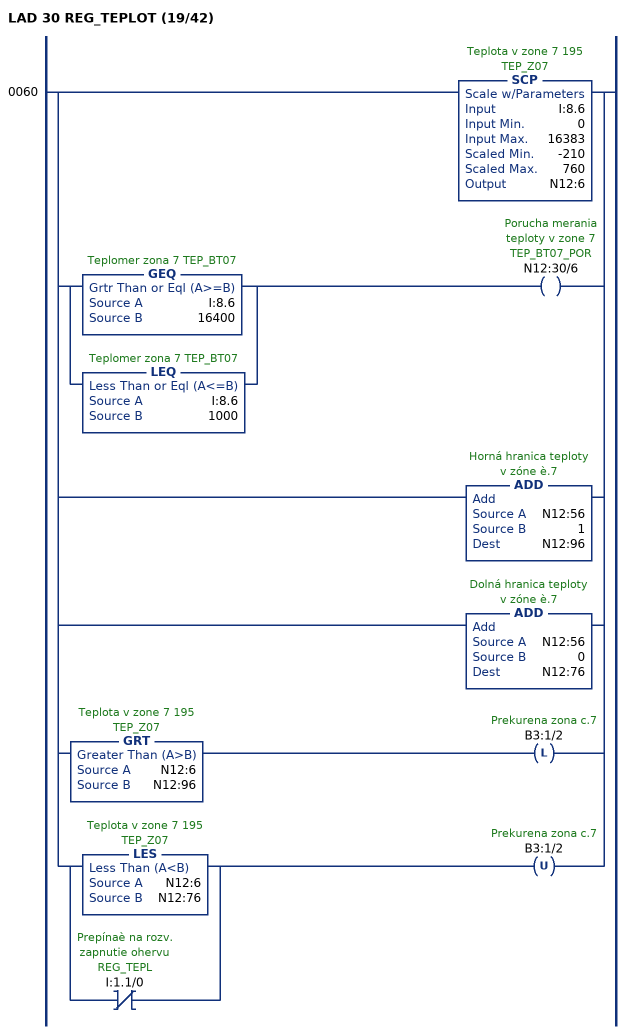
% Rung: 60 %
SOR BST SCP I:8.6 0 16383 -210 760 N12:6 NXB BST GEQ I:8.6 16400 NXB LEQ I:8.6 1000 BND OTE N12:30/6 NXB ADD N12:56 1 N12:96 NXB ADD N12:56 0 N12:76 NXB GRT N12:6 N12:96 OTL B3:1/2 NXB BST LES N12:6 N12:76 NXB XIO I:1.1/0 BND OTU B3:1/2 BND EOR
%   I:8.6  TEP_BT07  "Teplomer zona 7" %
%   N12:6  TEP_Z07  "Teplota v zone 7 195" %
%   N12:30/6  TEP_BT07_POR  "Porucha merania teploty v zone 7" %
%   N12:56  "Žiadaná teplota v zóne è.7" %
%   N12:96  "Horná hranica teploty v zóne è.7" %
%   N12:76  "Dolná hranica teploty v zóne è.7" %
%   B3:1/2  "Prekurena zona c.7" %
%   I:1.1/0  REG_TEPL  "Prepínaè na rozv. zapnutie ohervu" %

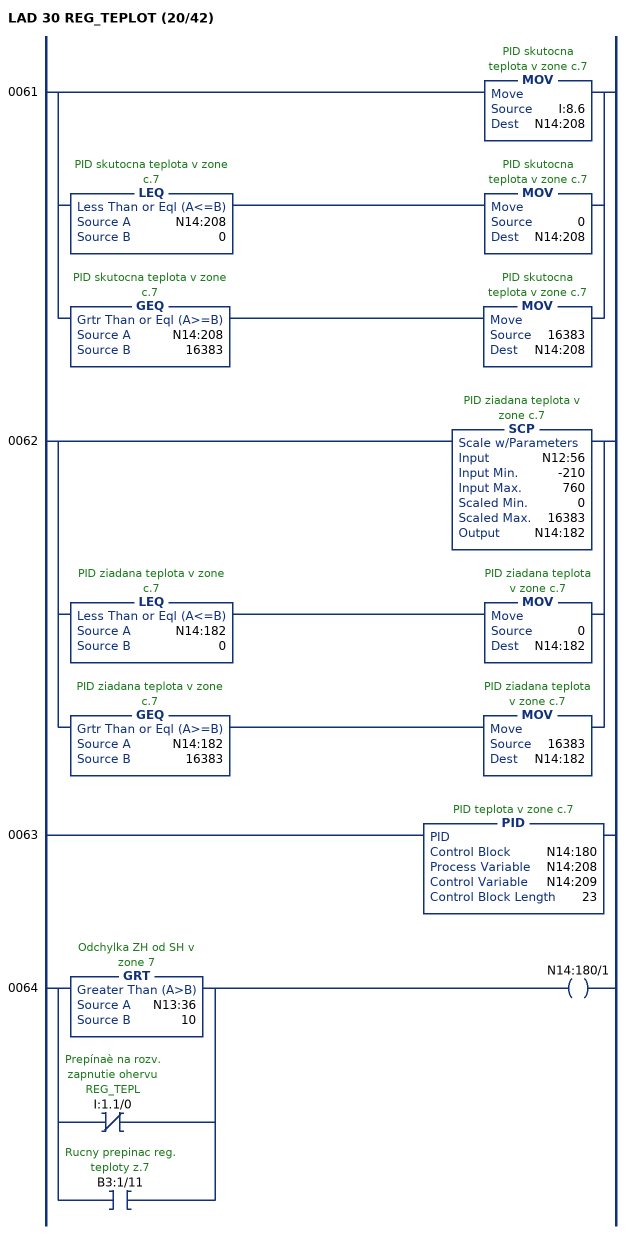
% Rung: 61 %
SOR BST MOV I:8.6 N14:208 NXB LEQ N14:208 0 MOV 0 N14:208 NXB GEQ N14:208 16383 MOV 16383 N14:208 BND EOR
%   I:8.6  TEP_BT07  "Teplomer zona 7" %
%   N14:208  "PID skutocna teplota v zone c.7" %
% Rung: 62 %
SOR BST SCP N12:56 -210 760 0 16383 N14:182 NXB LEQ N14:182 0 MOV 0 N14:182 NXB GEQ N14:182 16383 MOV 16383 N14:182 BND EOR
%   N12:56  "Žiadaná teplota v zóne è.7" %
%   N14:182  "PID ziadana teplota v zone c.7" %
% Rung: 63 %
SOR PID N14:180 N14:208 N14:209 23 EOR
%   N14:180  "PID teplota v zone c.7" %
%   N14:208  "PID skutocna teplota v zone c.7" %
% Rung: 64 %
SOR BST GRT N13:36 10 NXB XIO I:1.1/0 NXB XIC B3:1/11 BND OTE N14:180/1 EOR
%   N13:36  "Odchylka ZH od SH v zone 7" %
%   I:1.1/0  REG_TEPL  "Prepínaè na rozv. zapnutie ohervu" %
%   B3:1/11  "Rucny prepinac reg. teploty z.7" %

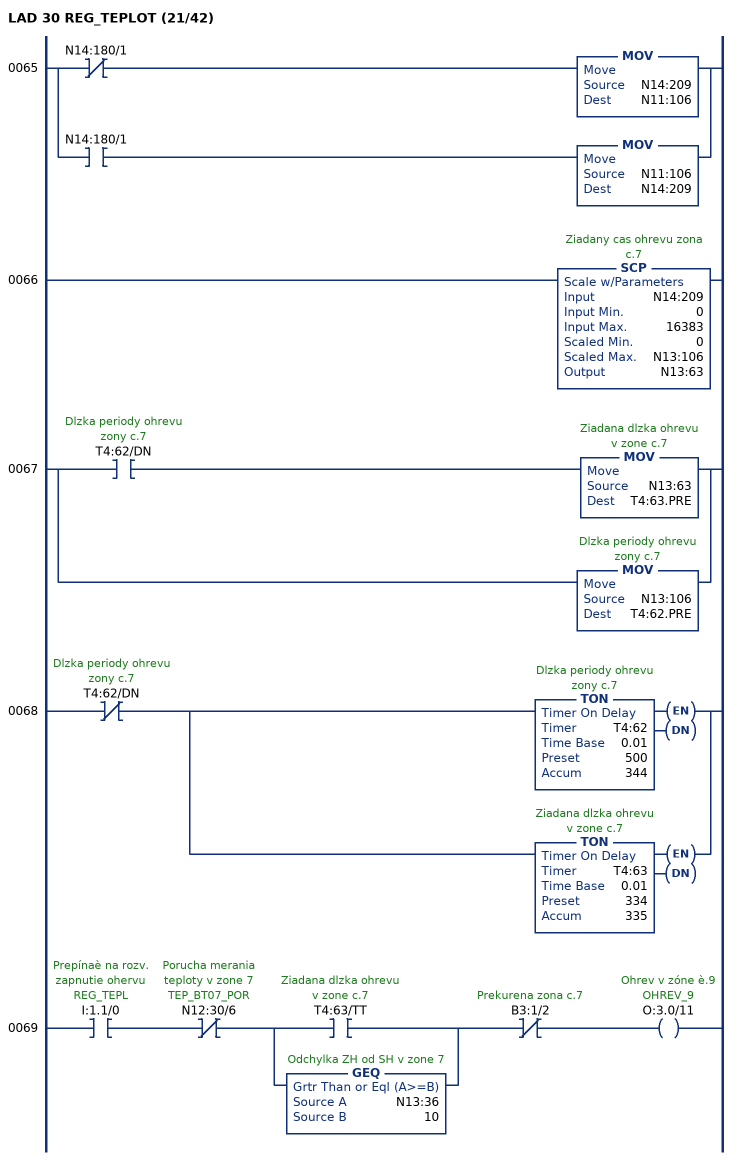
% Rung: 65 %
SOR BST XIO N14:180/1 MOV N14:209 N11:106 NXB XIC N14:180/1 MOV N11:106 N14:209 BND EOR
% Rung: 66 %
SOR SCP N14:209 0 16383 0 N13:106 N13:63 EOR
%   N13:63  "Ziadany cas ohrevu zona c.7" %
% Rung: 67 %
SOR BST XIC T4:62/DN MOV N13:63 T4:63.PRE NXB MOV N13:106 T4:62.PRE BND EOR
%   T4:62  "Dlzka periody ohrevu zony c.7" %
%   N13:63  "Ziadany cas ohrevu zona c.7" %
%   T4:63  "Ziadana dlzka ohrevu v zone c.7" %
% Rung: 68 %
SOR XIO T4:62/DN BST TON T4:62 0.01 500 344 NXB TON T4:63 0.01 334 335 BND EOR
%   T4:62  "Dlzka periody ohrevu zony c.7" %
%   T4:63  "Ziadana dlzka ohrevu v zone c.7" %
% Rung: 69 %
SOR XIC I:1.1/0 XIO N12:30/6 BST XIC T4:63/TT NXB GEQ N13:36 10 BND XIO B3:1/2 OTE O:3.0/11 EOR
%   I:1.1/0  REG_TEPL  "Prepínaè na rozv. zapnutie ohervu" %
%   N12:30/6  TEP_BT07_POR  "Porucha merania teploty v zone 7" %
%   T4:63  "Ziadana dlzka ohrevu v zone c.7" %
%   N13:36  "Odchylka ZH od SH v zone 7" %
%   B3:1/2  "Prekurena zona c.7" %
%   O:3.0/11  OHREV_9  "Ohrev v zóne è.9" %

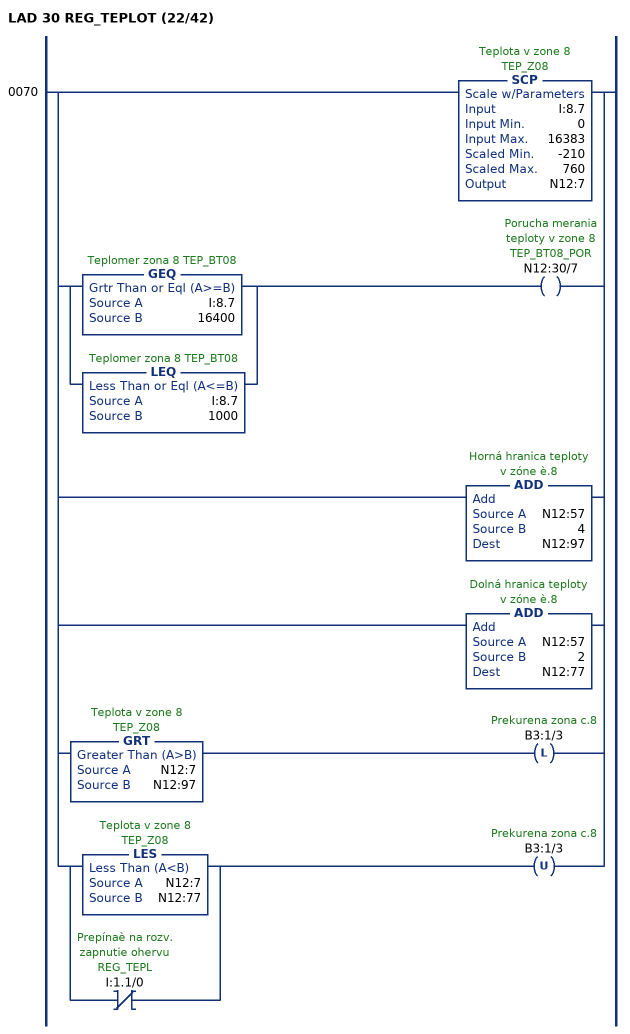
% Rung: 70 %
SOR BST SCP I:8.7 0 16383 -210 760 N12:7 NXB BST GEQ I:8.7 16400 NXB LEQ I:8.7 1000 BND OTE N12:30/7 NXB ADD N12:57 4 N12:97 NXB ADD N12:57 2 N12:77 NXB GRT N12:7 N12:97 OTL B3:1/3 NXB BST LES N12:7 N12:77 NXB XIO I:1.1/0 BND OTU B3:1/3 BND EOR
%   I:8.7  TEP_BT08  "Teplomer zona 8" %
%   N12:7  TEP_Z08  "Teplota v zone 8" %
%   N12:30/7  TEP_BT08_POR  "Porucha merania teploty v zone 8" %
%   N12:57  "Žiadaná teplota v zóne è.8" %
%   N12:97  "Horná hranica teploty v zóne è.8" %
%   N12:77  "Dolná hranica teploty v zóne è.8" %
%   B3:1/3  "Prekurena zona c.8" %
%   I:1.1/0  REG_TEPL  "Prepínaè na rozv. zapnutie ohervu" %

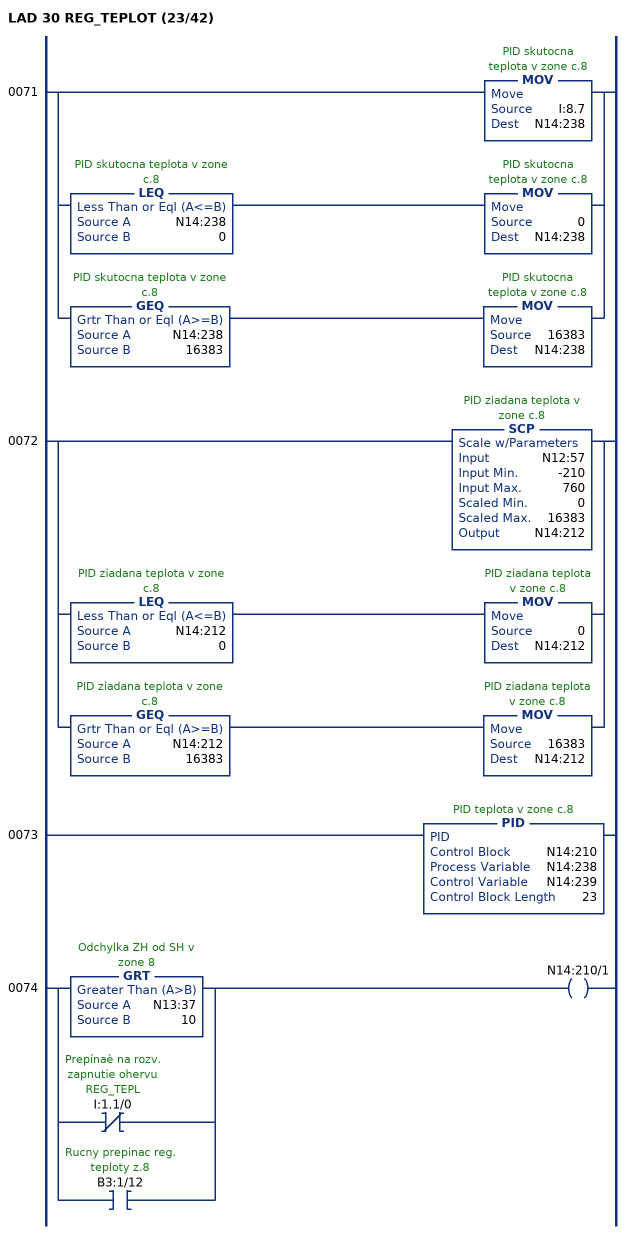
% Rung: 71 %
SOR BST MOV I:8.7 N14:238 NXB LEQ N14:238 0 MOV 0 N14:238 NXB GEQ N14:238 16383 MOV 16383 N14:238 BND EOR
%   I:8.7  TEP_BT08  "Teplomer zona 8" %
%   N14:238  "PID skutocna teplota v zone c.8" %
% Rung: 72 %
SOR BST SCP N12:57 -210 760 0 16383 N14:212 NXB LEQ N14:212 0 MOV 0 N14:212 NXB GEQ N14:212 16383 MOV 16383 N14:212 BND EOR
%   N12:57  "Žiadaná teplota v zóne è.8" %
%   N14:212  "PID ziadana teplota v zone c.8" %
% Rung: 73 %
SOR PID N14:210 N14:238 N14:239 23 EOR
%   N14:210  "PID teplota v zone c.8" %
%   N14:238  "PID skutocna teplota v zone c.8" %
% Rung: 74 %
SOR BST GRT N13:37 10 NXB XIO I:1.1/0 NXB XIC B3:1/12 BND OTE N14:210/1 EOR
%   N13:37  "Odchylka ZH od SH v zone 8" %
%   I:1.1/0  REG_TEPL  "Prepínaè na rozv. zapnutie ohervu" %
%   B3:1/12  "Rucny prepinac reg. teploty z.8" %

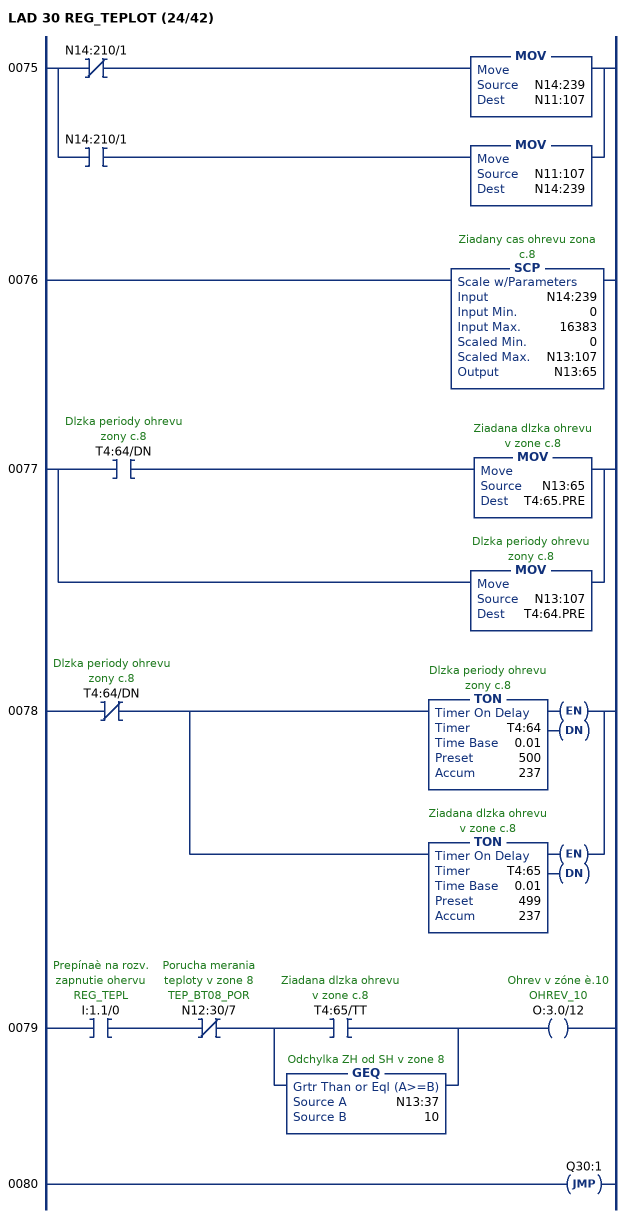
% Rung: 75 %
SOR BST XIO N14:210/1 MOV N14:239 N11:107 NXB XIC N14:210/1 MOV N11:107 N14:239 BND EOR
% Rung: 76 %
SOR SCP N14:239 0 16383 0 N13:107 N13:65 EOR
%   N13:65  "Ziadany cas ohrevu zona c.8" %
% Rung: 77 %
SOR BST XIC T4:64/DN MOV N13:65 T4:65.PRE NXB MOV N13:107 T4:64.PRE BND EOR
%   T4:64  "Dlzka periody ohrevu zony c.8" %
%   N13:65  "Ziadany cas ohrevu zona c.8" %
%   T4:65  "Ziadana dlzka ohrevu v zone c.8" %
% Rung: 78 %
SOR XIO T4:64/DN BST TON T4:64 0.01 500 237 NXB TON T4:65 0.01 499 237 BND EOR
%   T4:64  "Dlzka periody ohrevu zony c.8" %
%   T4:65  "Ziadana dlzka ohrevu v zone c.8" %
% Rung: 79 %
SOR XIC I:1.1/0 XIO N12:30/7 BST XIC T4:65/TT NXB GEQ N13:37 10 BND OTE O:3.0/12 EOR
%   I:1.1/0  REG_TEPL  "Prepínaè na rozv. zapnutie ohervu" %
%   N12:30/7  TEP_BT08_POR  "Porucha merania teploty v zone 8" %
%   T4:65  "Ziadana dlzka ohrevu v zone c.8" %
%   N13:37  "Odchylka ZH od SH v zone 8" %
%   O:3.0/12  OHREV_10  "Ohrev v zóne è.10" %
% Rung: 80 %
SOR JMP Q30:1 EOR

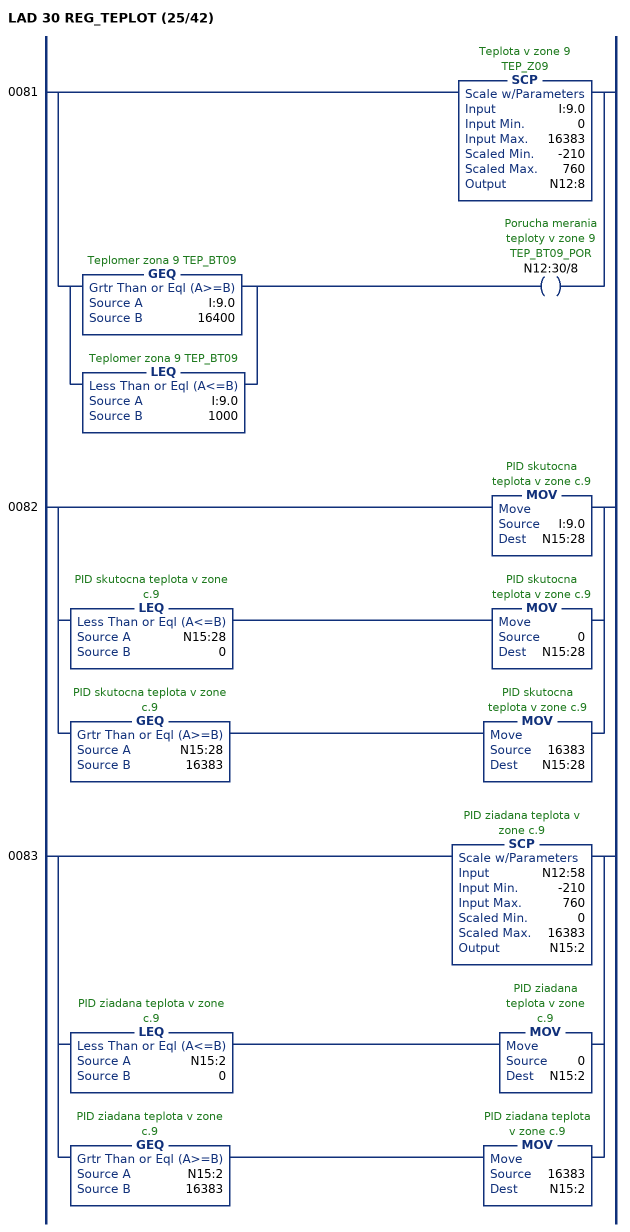
% Rung: 81 %
SOR BST SCP I:9.0 0 16383 -210 760 N12:8 NXB BST GEQ I:9.0 16400 NXB LEQ I:9.0 1000 BND OTE N12:30/8 BND EOR
%   I:9.0  TEP_BT09  "Teplomer zona 9" %
%   N12:8  TEP_Z09  "Teplota v zone 9" %
%   N12:30/8  TEP_BT09_POR  "Porucha merania teploty v zone 9" %
% Rung: 82 %
SOR BST MOV I:9.0 N15:28 NXB LEQ N15:28 0 MOV 0 N15:28 NXB GEQ N15:28 16383 MOV 16383 N15:28 BND EOR
%   I:9.0  TEP_BT09  "Teplomer zona 9" %
%   N15:28  "PID skutocna teplota v zone c.9" %
% Rung: 83 %
SOR BST SCP N12:58 -210 760 0 16383 N15:2 NXB LEQ N15:2 0 MOV 0 N15:2 NXB GEQ N15:2 16383 MOV 16383 N15:2 BND EOR
%   N12:58  "Žiadaná teplota v zóne è.9" %
%   N15:2  "PID ziadana teplota v zone c.9" %

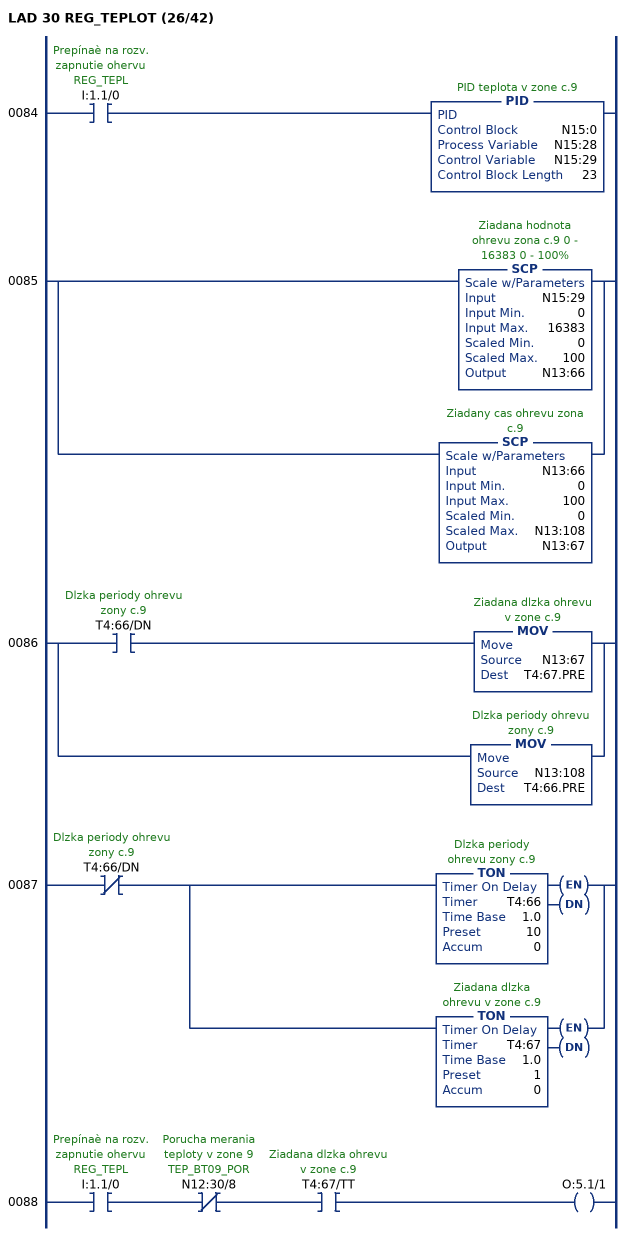
% Rung: 84 %
SOR XIC I:1.1/0 PID N15:0 N15:28 N15:29 23 EOR
%   I:1.1/0  REG_TEPL  "Prepínaè na rozv. zapnutie ohervu" %
%   N15:0  "PID teplota v zone c.9" %
%   N15:28  "PID skutocna teplota v zone c.9" %
% Rung: 85 %
SOR BST SCP N15:29 0 16383 0 100 N13:66 NXB SCP N13:66 0 100 0 N13:108 N13:67 BND EOR
%   N13:66  "Ziadana hodnota ohrevu zona c.9 0 - 16383 0 - 100%" %
%   N13:67  "Ziadany cas ohrevu zona c.9" %
% Rung: 86 %
SOR BST XIC T4:66/DN MOV N13:67 T4:67.PRE NXB MOV N13:108 T4:66.PRE BND EOR
%   T4:66  "Dlzka periody ohrevu zony c.9" %
%   N13:67  "Ziadany cas ohrevu zona c.9" %
%   T4:67  "Ziadana dlzka ohrevu v zone c.9" %
% Rung: 87 %
SOR XIO T4:66/DN BST TON T4:66 1.0 10 0 NXB TON T4:67 1.0 1 0 BND EOR
%   T4:66  "Dlzka periody ohrevu zony c.9" %
%   T4:67  "Ziadana dlzka ohrevu v zone c.9" %
% Rung: 88 %
SOR XIC I:1.1/0 XIO N12:30/8 XIC T4:67/TT OTE O:5.1/1 EOR
%   I:1.1/0  REG_TEPL  "Prepínaè na rozv. zapnutie ohervu" %
%   N12:30/8  TEP_BT09_POR  "Porucha merania teploty v zone 9" %
%   T4:67  "Ziadana dlzka ohrevu v zone c.9" %

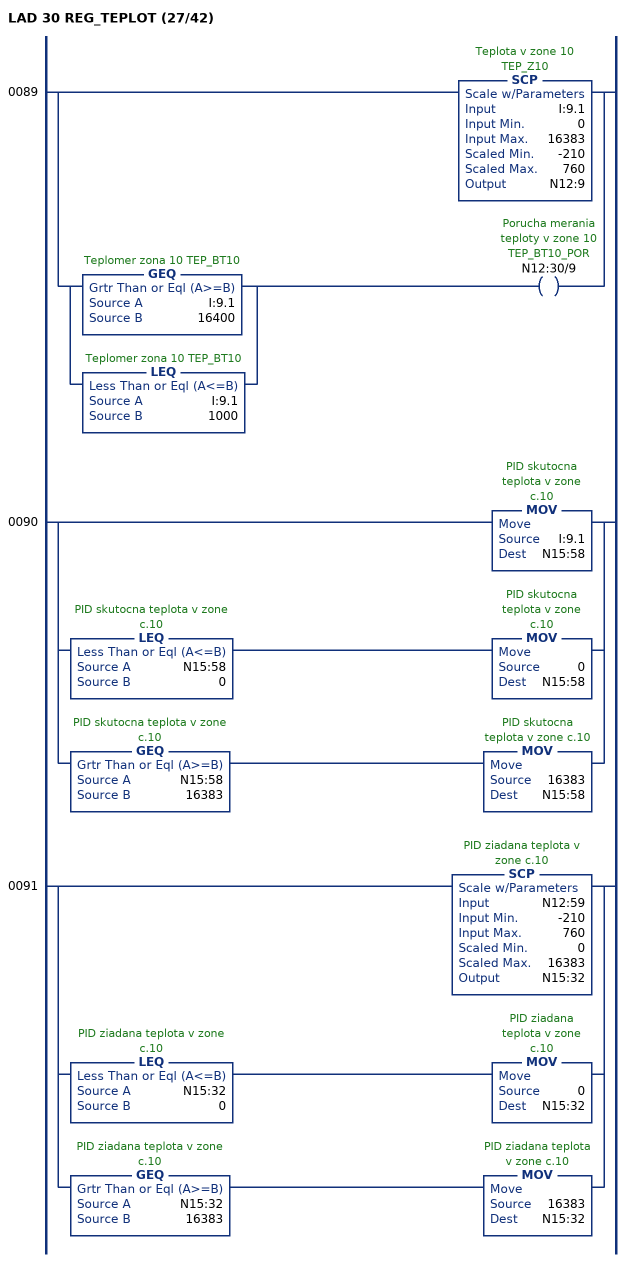
% Rung: 89 %
SOR BST SCP I:9.1 0 16383 -210 760 N12:9 NXB BST GEQ I:9.1 16400 NXB LEQ I:9.1 1000 BND OTE N12:30/9 BND EOR
%   I:9.1  TEP_BT10  "Teplomer zona 10" %
%   N12:9  TEP_Z10  "Teplota v zone 10" %
%   N12:30/9  TEP_BT10_POR  "Porucha merania teploty v zone 10" %
% Rung: 90 %
SOR BST MOV I:9.1 N15:58 NXB LEQ N15:58 0 MOV 0 N15:58 NXB GEQ N15:58 16383 MOV 16383 N15:58 BND EOR
%   I:9.1  TEP_BT10  "Teplomer zona 10" %
%   N15:58  "PID skutocna teplota v zone c.10" %
% Rung: 91 %
SOR BST SCP N12:59 -210 760 0 16383 N15:32 NXB LEQ N15:32 0 MOV 0 N15:32 NXB GEQ N15:32 16383 MOV 16383 N15:32 BND EOR
%   N12:59  "Žiadaná teplota v zóne è.10" %
%   N15:32  "PID ziadana teplota v zone c.10" %

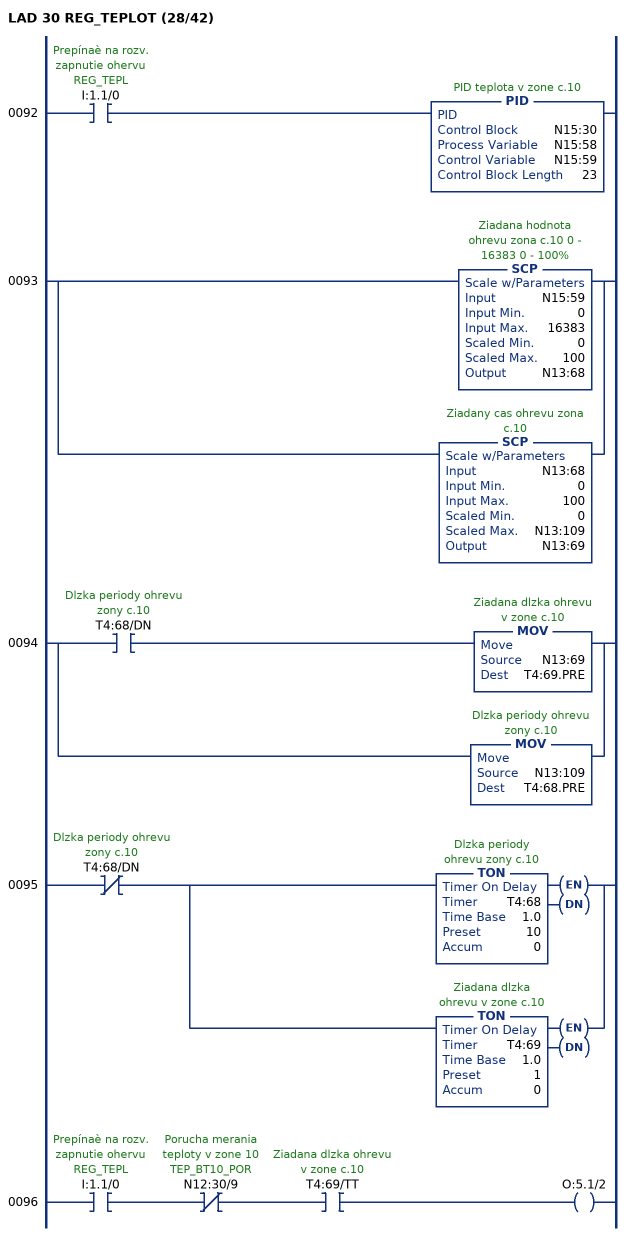
% Rung: 92 %
SOR XIC I:1.1/0 PID N15:30 N15:58 N15:59 23 EOR
%   I:1.1/0  REG_TEPL  "Prepínaè na rozv. zapnutie ohervu" %
%   N15:30  "PID teplota v zone c.10" %
%   N15:58  "PID skutocna teplota v zone c.10" %
% Rung: 93 %
SOR BST SCP N15:59 0 16383 0 100 N13:68 NXB SCP N13:68 0 100 0 N13:109 N13:69 BND EOR
%   N13:68  "Ziadana hodnota ohrevu zona c.10 0 - 16383 0 - 100%" %
%   N13:69  "Ziadany cas ohrevu zona c.10" %
% Rung: 94 %
SOR BST XIC T4:68/DN MOV N13:69 T4:69.PRE NXB MOV N13:109 T4:68.PRE BND EOR
%   T4:68  "Dlzka periody ohrevu zony c.10" %
%   N13:69  "Ziadany cas ohrevu zona c.10" %
%   T4:69  "Ziadana dlzka ohrevu v zone c.10" %
% Rung: 95 %
SOR XIO T4:68/DN BST TON T4:68 1.0 10 0 NXB TON T4:69 1.0 1 0 BND EOR
%   T4:68  "Dlzka periody ohrevu zony c.10" %
%   T4:69  "Ziadana dlzka ohrevu v zone c.10" %
% Rung: 96 %
SOR XIC I:1.1/0 XIO N12:30/9 XIC T4:69/TT OTE O:5.1/2 EOR
%   I:1.1/0  REG_TEPL  "Prepínaè na rozv. zapnutie ohervu" %
%   N12:30/9  TEP_BT10_POR  "Porucha merania teploty v zone 10" %
%   T4:69  "Ziadana dlzka ohrevu v zone c.10" %

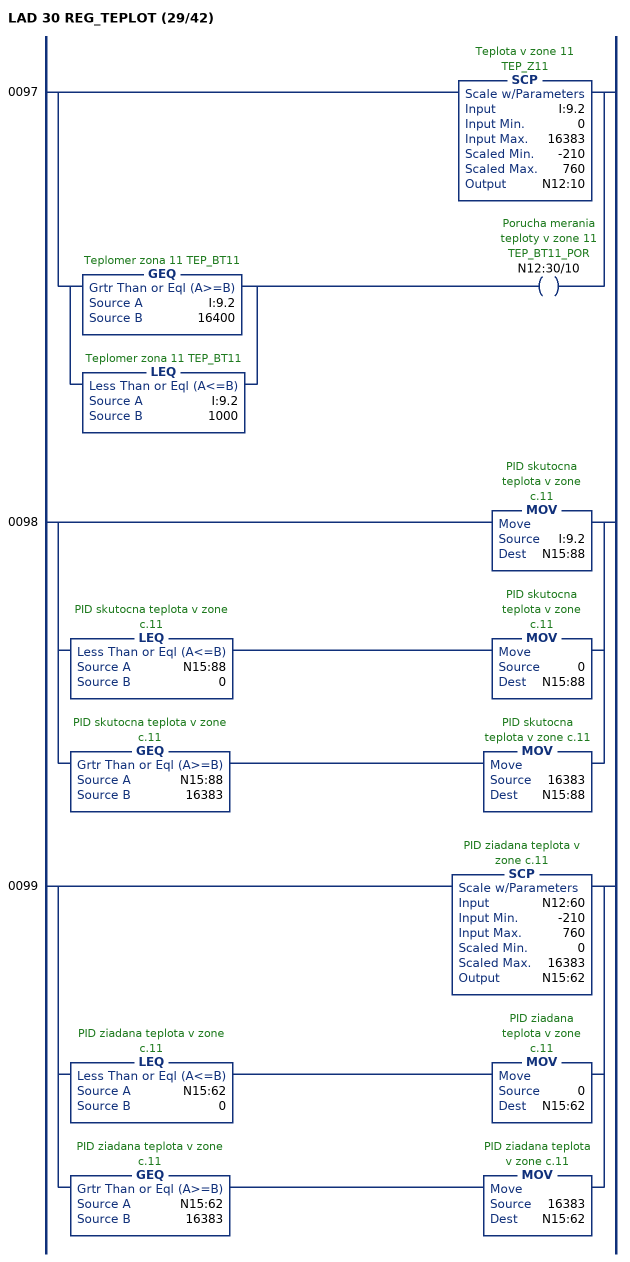
% Rung: 97 %
SOR BST SCP I:9.2 0 16383 -210 760 N12:10 NXB BST GEQ I:9.2 16400 NXB LEQ I:9.2 1000 BND OTE N12:30/10 BND EOR
%   I:9.2  TEP_BT11  "Teplomer zona 11" %
%   N12:10  TEP_Z11  "Teplota v zone 11" %
%   N12:30/10  TEP_BT11_POR  "Porucha merania teploty v zone 11" %
% Rung: 98 %
SOR BST MOV I:9.2 N15:88 NXB LEQ N15:88 0 MOV 0 N15:88 NXB GEQ N15:88 16383 MOV 16383 N15:88 BND EOR
%   I:9.2  TEP_BT11  "Teplomer zona 11" %
%   N15:88  "PID skutocna teplota v zone c.11" %
% Rung: 99 %
SOR BST SCP N12:60 -210 760 0 16383 N15:62 NXB LEQ N15:62 0 MOV 0 N15:62 NXB GEQ N15:62 16383 MOV 16383 N15:62 BND EOR
%   N12:60  "Žiadaná teplota v zóne è.11" %
%   N15:62  "PID ziadana teplota v zone c.11" %

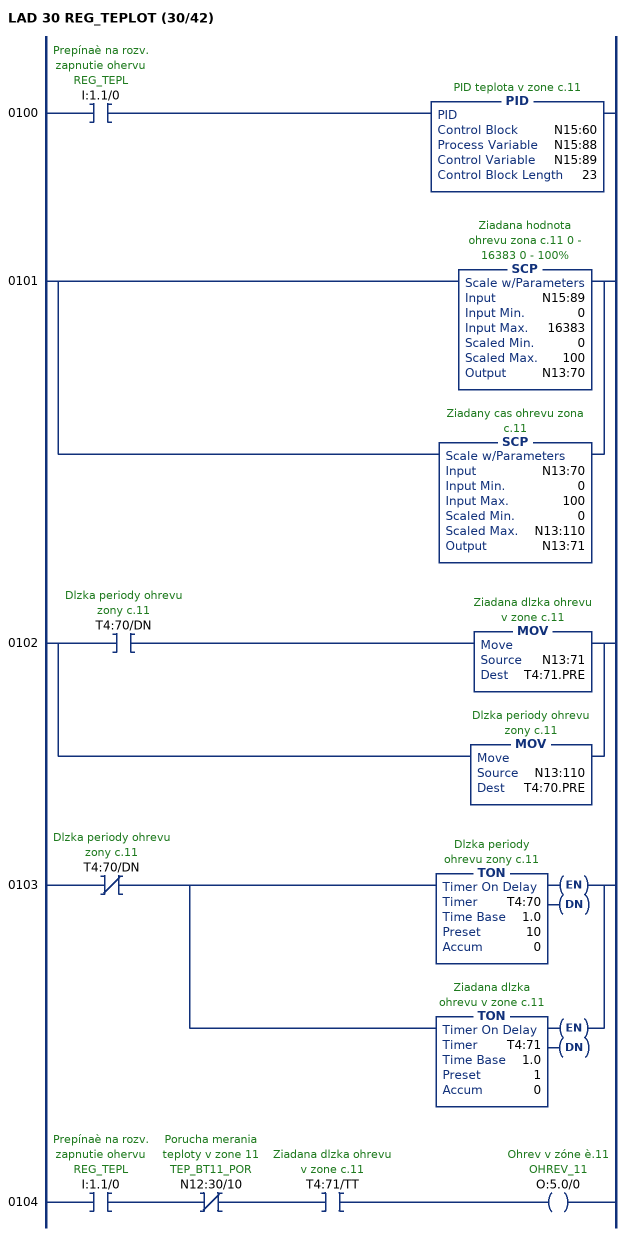
% Rung: 100 %
SOR XIC I:1.1/0 PID N15:60 N15:88 N15:89 23 EOR
%   I:1.1/0  REG_TEPL  "Prepínaè na rozv. zapnutie ohervu" %
%   N15:60  "PID teplota v zone c.11" %
%   N15:88  "PID skutocna teplota v zone c.11" %
% Rung: 101 %
SOR BST SCP N15:89 0 16383 0 100 N13:70 NXB SCP N13:70 0 100 0 N13:110 N13:71 BND EOR
%   N13:70  "Ziadana hodnota ohrevu zona c.11 0 - 16383 0 - 100%" %
%   N13:71  "Ziadany cas ohrevu zona c.11" %
% Rung: 102 %
SOR BST XIC T4:70/DN MOV N13:71 T4:71.PRE NXB MOV N13:110 T4:70.PRE BND EOR
%   T4:70  "Dlzka periody ohrevu zony c.11" %
%   N13:71  "Ziadany cas ohrevu zona c.11" %
%   T4:71  "Ziadana dlzka ohrevu v zone c.11" %
% Rung: 103 %
SOR XIO T4:70/DN BST TON T4:70 1.0 10 0 NXB TON T4:71 1.0 1 0 BND EOR
%   T4:70  "Dlzka periody ohrevu zony c.11" %
%   T4:71  "Ziadana dlzka ohrevu v zone c.11" %
% Rung: 104 %
SOR XIC I:1.1/0 XIO N12:30/10 XIC T4:71/TT OTE O:5.0/0 EOR
%   I:1.1/0  REG_TEPL  "Prepínaè na rozv. zapnutie ohervu" %
%   N12:30/10  TEP_BT11_POR  "Porucha merania teploty v zone 11" %
%   T4:71  "Ziadana dlzka ohrevu v zone c.11" %
%   O:5.0/0  OHREV_11  "Ohrev v zóne è.11" %

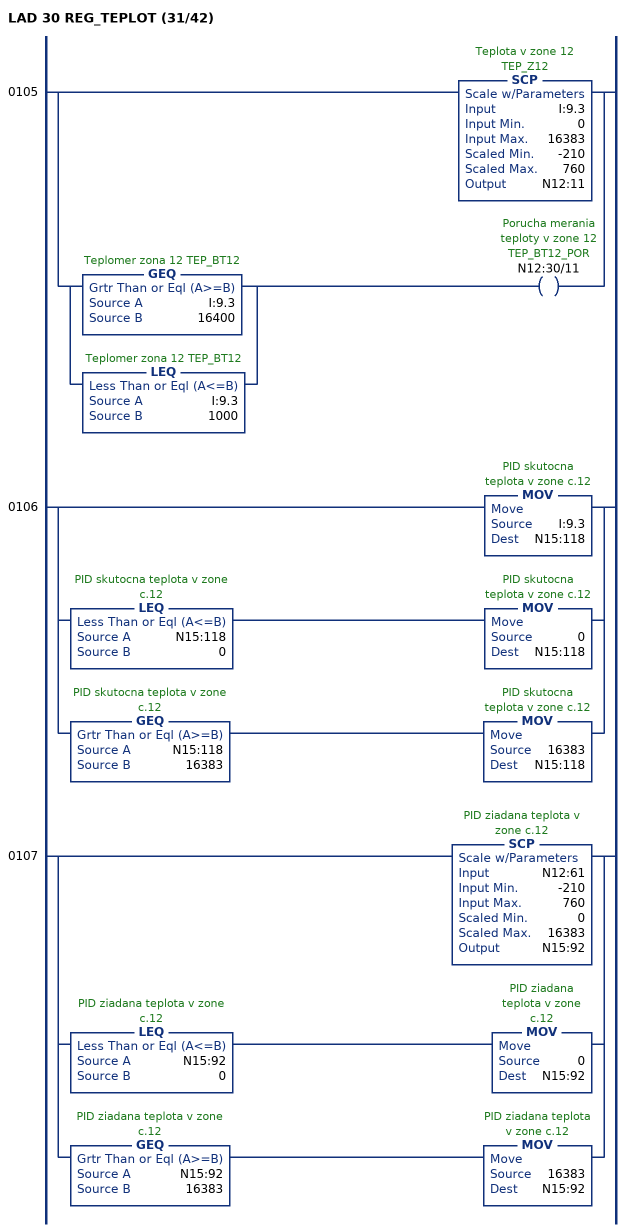
% Rung: 105 %
SOR BST SCP I:9.3 0 16383 -210 760 N12:11 NXB BST GEQ I:9.3 16400 NXB LEQ I:9.3 1000 BND OTE N12:30/11 BND EOR
%   I:9.3  TEP_BT12  "Teplomer zona 12" %
%   N12:11  TEP_Z12  "Teplota v zone 12" %
%   N12:30/11  TEP_BT12_POR  "Porucha merania teploty v zone 12" %
% Rung: 106 %
SOR BST MOV I:9.3 N15:118 NXB LEQ N15:118 0 MOV 0 N15:118 NXB GEQ N15:118 16383 MOV 16383 N15:118 BND EOR
%   I:9.3  TEP_BT12  "Teplomer zona 12" %
%   N15:118  "PID skutocna teplota v zone c.12" %
% Rung: 107 %
SOR BST SCP N12:61 -210 760 0 16383 N15:92 NXB LEQ N15:92 0 MOV 0 N15:92 NXB GEQ N15:92 16383 MOV 16383 N15:92 BND EOR
%   N12:61  "Žiadaná teplota v zóne è.12" %
%   N15:92  "PID ziadana teplota v zone c.12" %

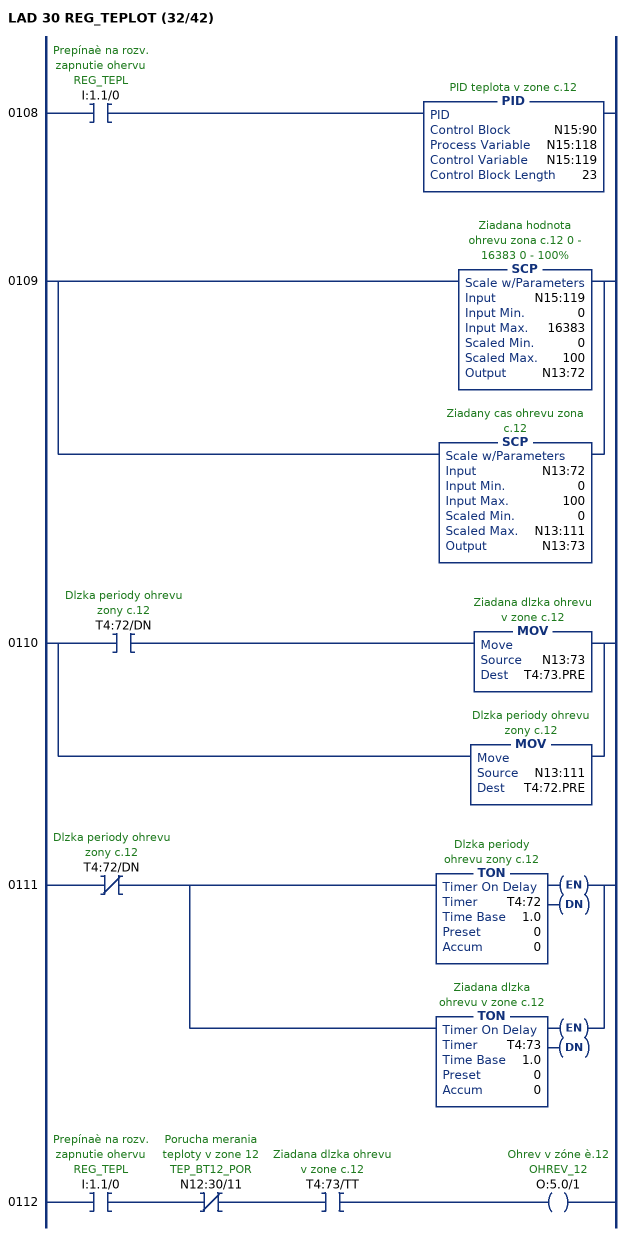
% Rung: 108 %
SOR XIC I:1.1/0 PID N15:90 N15:118 N15:119 23 EOR
%   I:1.1/0  REG_TEPL  "Prepínaè na rozv. zapnutie ohervu" %
%   N15:90  "PID teplota v zone c.12" %
%   N15:118  "PID skutocna teplota v zone c.12" %
% Rung: 109 %
SOR BST SCP N15:119 0 16383 0 100 N13:72 NXB SCP N13:72 0 100 0 N13:111 N13:73 BND EOR
%   N13:72  "Ziadana hodnota ohrevu zona c.12 0 - 16383 0 - 100%" %
%   N13:73  "Ziadany cas ohrevu zona c.12" %
% Rung: 110 %
SOR BST XIC T4:72/DN MOV N13:73 T4:73.PRE NXB MOV N13:111 T4:72.PRE BND EOR
%   T4:72  "Dlzka periody ohrevu zony c.12" %
%   N13:73  "Ziadany cas ohrevu zona c.12" %
%   T4:73  "Ziadana dlzka ohrevu v zone c.12" %
% Rung: 111 %
SOR XIO T4:72/DN BST TON T4:72 1.0 0 0 NXB TON T4:73 1.0 0 0 BND EOR
%   T4:72  "Dlzka periody ohrevu zony c.12" %
%   T4:73  "Ziadana dlzka ohrevu v zone c.12" %
% Rung: 112 %
SOR XIC I:1.1/0 XIO N12:30/11 XIC T4:73/TT OTE O:5.0/1 EOR
%   I:1.1/0  REG_TEPL  "Prepínaè na rozv. zapnutie ohervu" %
%   N12:30/11  TEP_BT12_POR  "Porucha merania teploty v zone 12" %
%   T4:73  "Ziadana dlzka ohrevu v zone c.12" %
%   O:5.0/1  OHREV_12  "Ohrev v zóne è.12" %

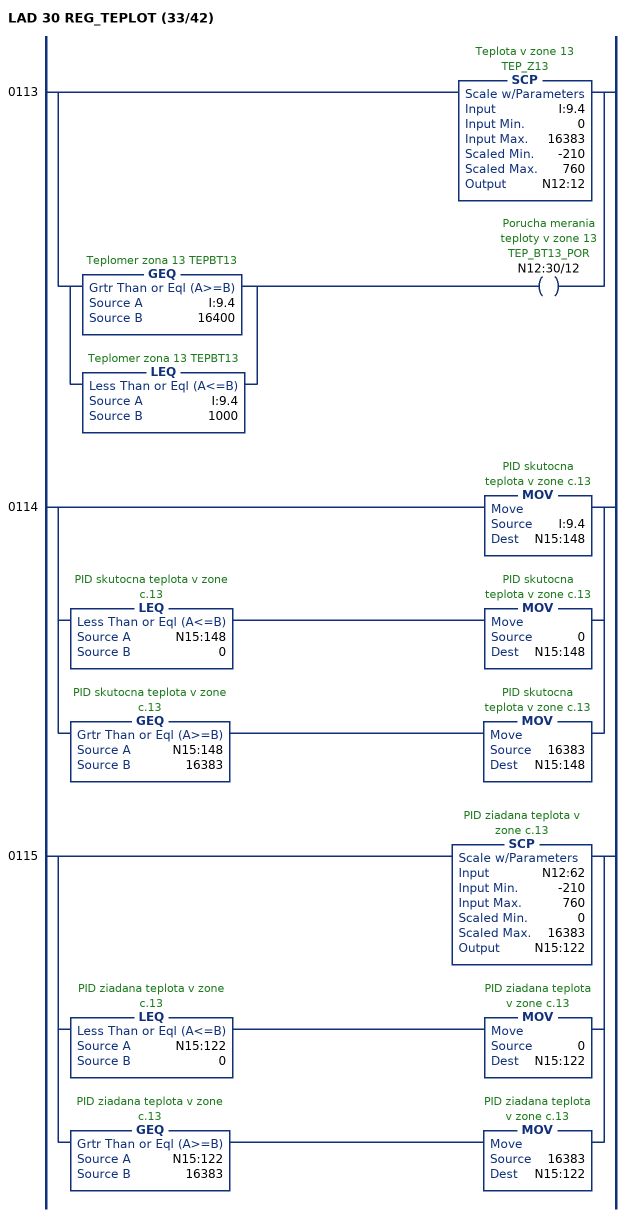
% Rung: 113 %
SOR BST SCP I:9.4 0 16383 -210 760 N12:12 NXB BST GEQ I:9.4 16400 NXB LEQ I:9.4 1000 BND OTE N12:30/12 BND EOR
%   I:9.4  TEPBT13  "Teplomer zona 13" %
%   N12:12  TEP_Z13  "Teplota v zone 13" %
%   N12:30/12  TEP_BT13_POR  "Porucha merania teploty v zone 13" %
% Rung: 114 %
SOR BST MOV I:9.4 N15:148 NXB LEQ N15:148 0 MOV 0 N15:148 NXB GEQ N15:148 16383 MOV 16383 N15:148 BND EOR
%   I:9.4  TEPBT13  "Teplomer zona 13" %
%   N15:148  "PID skutocna teplota v zone c.13" %
% Rung: 115 %
SOR BST SCP N12:62 -210 760 0 16383 N15:122 NXB LEQ N15:122 0 MOV 0 N15:122 NXB GEQ N15:122 16383 MOV 16383 N15:122 BND EOR
%   N12:62  "Žiadaná teplota v zóne è.13" %
%   N15:122  "PID ziadana teplota v zone c.13" %

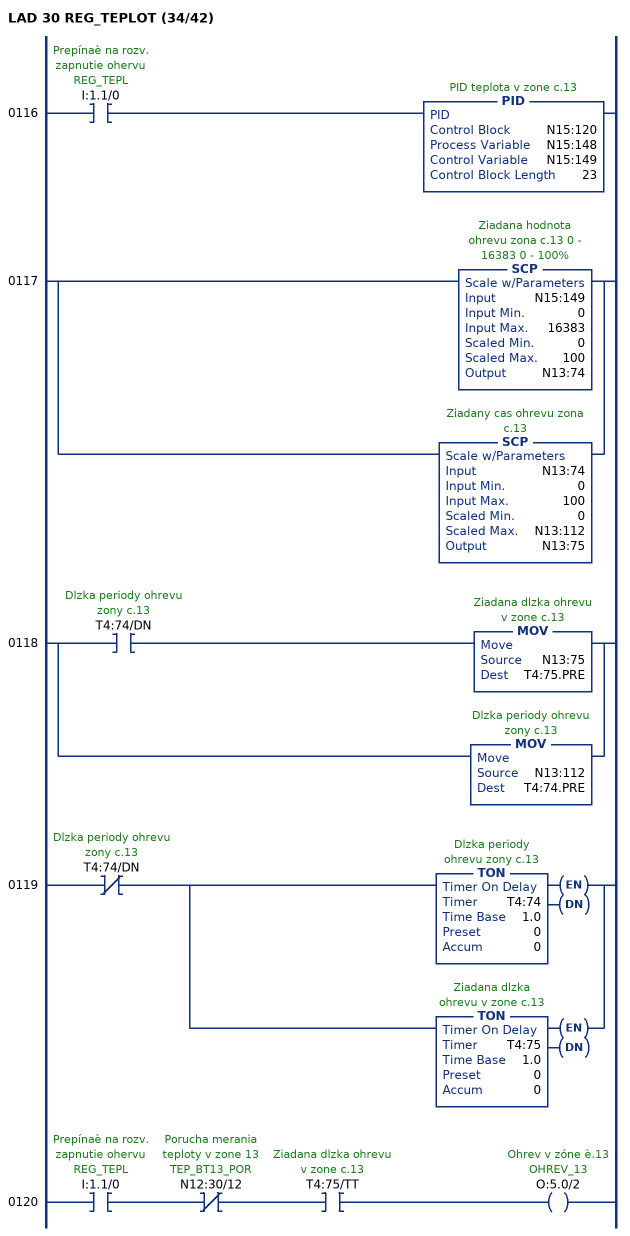
% Rung: 116 %
SOR XIC I:1.1/0 PID N15:120 N15:148 N15:149 23 EOR
%   I:1.1/0  REG_TEPL  "Prepínaè na rozv. zapnutie ohervu" %
%   N15:120  "PID teplota v zone c.13" %
%   N15:148  "PID skutocna teplota v zone c.13" %
% Rung: 117 %
SOR BST SCP N15:149 0 16383 0 100 N13:74 NXB SCP N13:74 0 100 0 N13:112 N13:75 BND EOR
%   N13:74  "Ziadana hodnota ohrevu zona c.13 0 - 16383 0 - 100%" %
%   N13:75  "Ziadany cas ohrevu zona c.13" %
% Rung: 118 %
SOR BST XIC T4:74/DN MOV N13:75 T4:75.PRE NXB MOV N13:112 T4:74.PRE BND EOR
%   T4:74  "Dlzka periody ohrevu zony c.13" %
%   N13:75  "Ziadany cas ohrevu zona c.13" %
%   T4:75  "Ziadana dlzka ohrevu v zone c.13" %
% Rung: 119 %
SOR XIO T4:74/DN BST TON T4:74 1.0 0 0 NXB TON T4:75 1.0 0 0 BND EOR
%   T4:74  "Dlzka periody ohrevu zony c.13" %
%   T4:75  "Ziadana dlzka ohrevu v zone c.13" %
% Rung: 120 %
SOR XIC I:1.1/0 XIO N12:30/12 XIC T4:75/TT OTE O:5.0/2 EOR
%   I:1.1/0  REG_TEPL  "Prepínaè na rozv. zapnutie ohervu" %
%   N12:30/12  TEP_BT13_POR  "Porucha merania teploty v zone 13" %
%   T4:75  "Ziadana dlzka ohrevu v zone c.13" %
%   O:5.0/2  OHREV_13  "Ohrev v zóne è.13" %

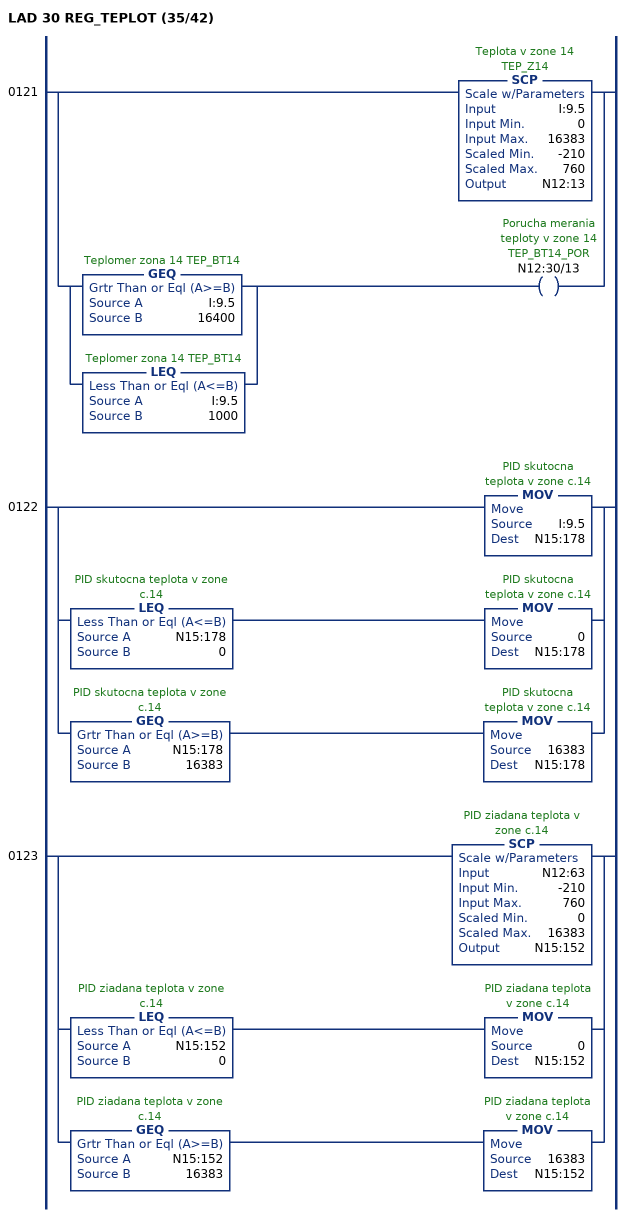
% Rung: 121 %
SOR BST SCP I:9.5 0 16383 -210 760 N12:13 NXB BST GEQ I:9.5 16400 NXB LEQ I:9.5 1000 BND OTE N12:30/13 BND EOR
%   I:9.5  TEP_BT14  "Teplomer zona 14" %
%   N12:13  TEP_Z14  "Teplota v zone 14" %
%   N12:30/13  TEP_BT14_POR  "Porucha merania teploty v zone 14" %
% Rung: 122 %
SOR BST MOV I:9.5 N15:178 NXB LEQ N15:178 0 MOV 0 N15:178 NXB GEQ N15:178 16383 MOV 16383 N15:178 BND EOR
%   I:9.5  TEP_BT14  "Teplomer zona 14" %
%   N15:178  "PID skutocna teplota v zone c.14" %
% Rung: 123 %
SOR BST SCP N12:63 -210 760 0 16383 N15:152 NXB LEQ N15:152 0 MOV 0 N15:152 NXB GEQ N15:152 16383 MOV 16383 N15:152 BND EOR
%   N12:63  "Žiadaná teplota v zóne è.14" %
%   N15:152  "PID ziadana teplota v zone c.14" %

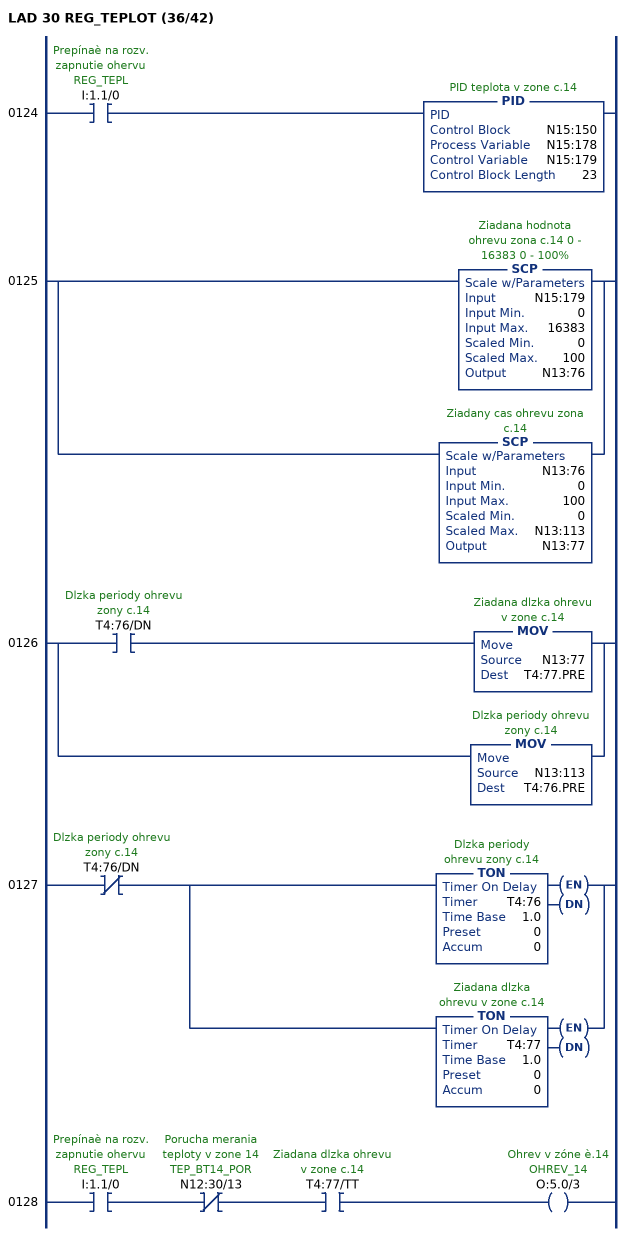
% Rung: 124 %
SOR XIC I:1.1/0 PID N15:150 N15:178 N15:179 23 EOR
%   I:1.1/0  REG_TEPL  "Prepínaè na rozv. zapnutie ohervu" %
%   N15:150  "PID teplota v zone c.14" %
%   N15:178  "PID skutocna teplota v zone c.14" %
% Rung: 125 %
SOR BST SCP N15:179 0 16383 0 100 N13:76 NXB SCP N13:76 0 100 0 N13:113 N13:77 BND EOR
%   N13:76  "Ziadana hodnota ohrevu zona c.14 0 - 16383 0 - 100%" %
%   N13:77  "Ziadany cas ohrevu zona c.14" %
% Rung: 126 %
SOR BST XIC T4:76/DN MOV N13:77 T4:77.PRE NXB MOV N13:113 T4:76.PRE BND EOR
%   T4:76  "Dlzka periody ohrevu zony c.14" %
%   N13:77  "Ziadany cas ohrevu zona c.14" %
%   T4:77  "Ziadana dlzka ohrevu v zone c.14" %
% Rung: 127 %
SOR XIO T4:76/DN BST TON T4:76 1.0 0 0 NXB TON T4:77 1.0 0 0 BND EOR
%   T4:76  "Dlzka periody ohrevu zony c.14" %
%   T4:77  "Ziadana dlzka ohrevu v zone c.14" %
% Rung: 128 %
SOR XIC I:1.1/0 XIO N12:30/13 XIC T4:77/TT OTE O:5.0/3 EOR
%   I:1.1/0  REG_TEPL  "Prepínaè na rozv. zapnutie ohervu" %
%   N12:30/13  TEP_BT14_POR  "Porucha merania teploty v zone 14" %
%   T4:77  "Ziadana dlzka ohrevu v zone c.14" %
%   O:5.0/3  OHREV_14  "Ohrev v zóne è.14" %

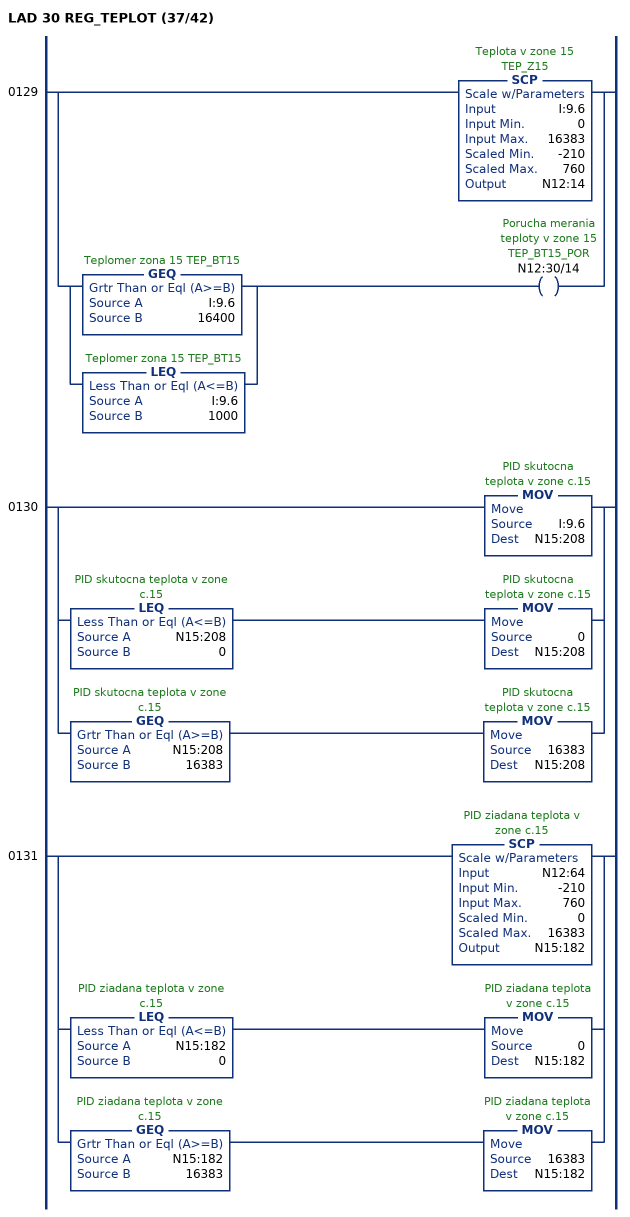
% Rung: 129 %
SOR BST SCP I:9.6 0 16383 -210 760 N12:14 NXB BST GEQ I:9.6 16400 NXB LEQ I:9.6 1000 BND OTE N12:30/14 BND EOR
%   I:9.6  TEP_BT15  "Teplomer zona 15" %
%   N12:14  TEP_Z15  "Teplota v zone 15" %
%   N12:30/14  TEP_BT15_POR  "Porucha merania teploty v zone 15" %
% Rung: 130 %
SOR BST MOV I:9.6 N15:208 NXB LEQ N15:208 0 MOV 0 N15:208 NXB GEQ N15:208 16383 MOV 16383 N15:208 BND EOR
%   I:9.6  TEP_BT15  "Teplomer zona 15" %
%   N15:208  "PID skutocna teplota v zone c.15" %
% Rung: 131 %
SOR BST SCP N12:64 -210 760 0 16383 N15:182 NXB LEQ N15:182 0 MOV 0 N15:182 NXB GEQ N15:182 16383 MOV 16383 N15:182 BND EOR
%   N12:64  "Žiadaná teplota v zóne è.15" %
%   N15:182  "PID ziadana teplota v zone c.15" %

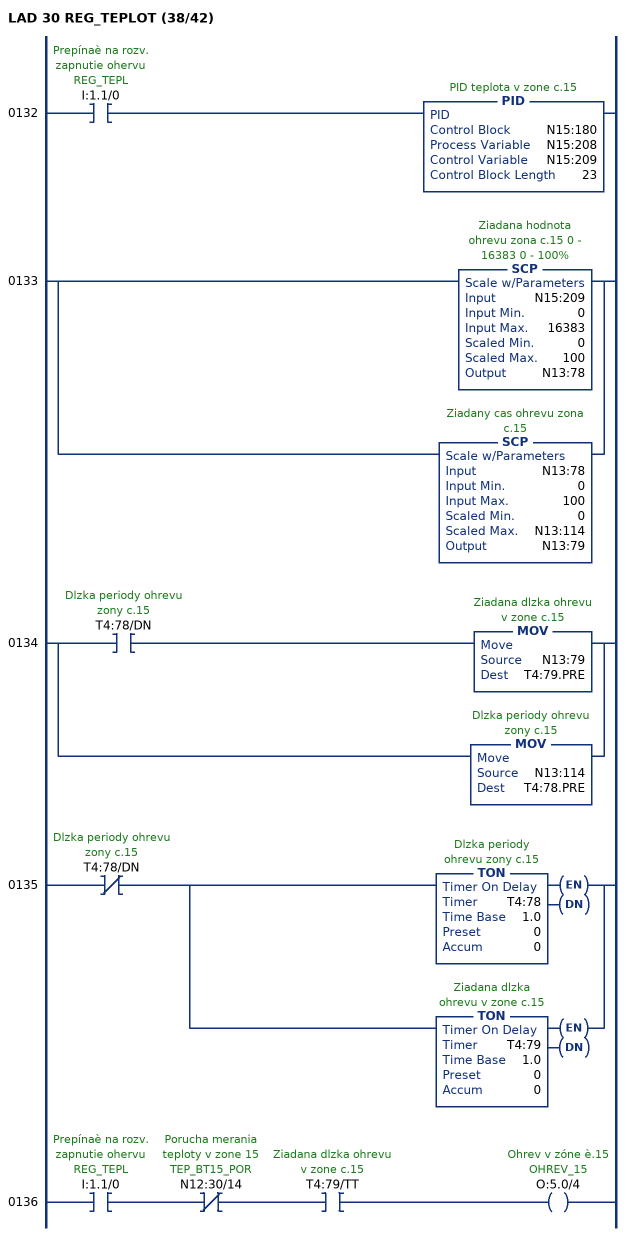
% Rung: 132 %
SOR XIC I:1.1/0 PID N15:180 N15:208 N15:209 23 EOR
%   I:1.1/0  REG_TEPL  "Prepínaè na rozv. zapnutie ohervu" %
%   N15:180  "PID teplota v zone c.15" %
%   N15:208  "PID skutocna teplota v zone c.15" %
% Rung: 133 %
SOR BST SCP N15:209 0 16383 0 100 N13:78 NXB SCP N13:78 0 100 0 N13:114 N13:79 BND EOR
%   N13:78  "Ziadana hodnota ohrevu zona c.15 0 - 16383 0 - 100%" %
%   N13:79  "Ziadany cas ohrevu zona c.15" %
% Rung: 134 %
SOR BST XIC T4:78/DN MOV N13:79 T4:79.PRE NXB MOV N13:114 T4:78.PRE BND EOR
%   T4:78  "Dlzka periody ohrevu zony c.15" %
%   N13:79  "Ziadany cas ohrevu zona c.15" %
%   T4:79  "Ziadana dlzka ohrevu v zone c.15" %
% Rung: 135 %
SOR XIO T4:78/DN BST TON T4:78 1.0 0 0 NXB TON T4:79 1.0 0 0 BND EOR
%   T4:78  "Dlzka periody ohrevu zony c.15" %
%   T4:79  "Ziadana dlzka ohrevu v zone c.15" %
% Rung: 136 %
SOR XIC I:1.1/0 XIO N12:30/14 XIC T4:79/TT OTE O:5.0/4 EOR
%   I:1.1/0  REG_TEPL  "Prepínaè na rozv. zapnutie ohervu" %
%   N12:30/14  TEP_BT15_POR  "Porucha merania teploty v zone 15" %
%   T4:79  "Ziadana dlzka ohrevu v zone c.15" %
%   O:5.0/4  OHREV_15  "Ohrev v zóne è.15" %

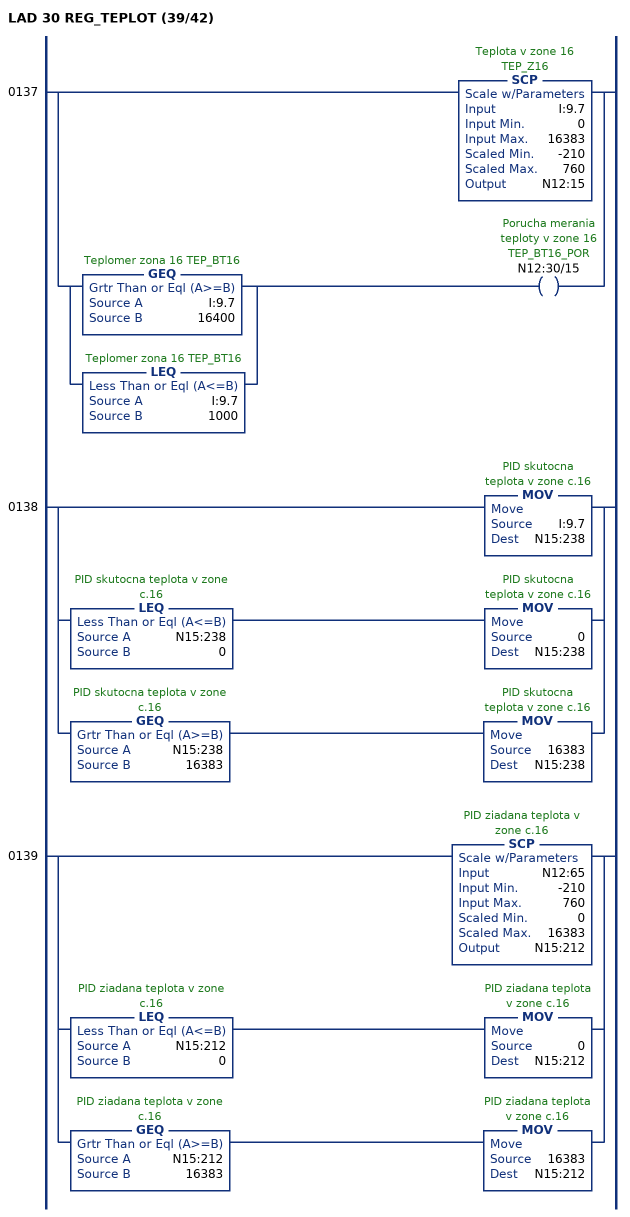
% Rung: 137 %
SOR BST SCP I:9.7 0 16383 -210 760 N12:15 NXB BST GEQ I:9.7 16400 NXB LEQ I:9.7 1000 BND OTE N12:30/15 BND EOR
%   I:9.7  TEP_BT16  "Teplomer zona 16" %
%   N12:15  TEP_Z16  "Teplota v zone 16" %
%   N12:30/15  TEP_BT16_POR  "Porucha merania teploty v zone 16" %
% Rung: 138 %
SOR BST MOV I:9.7 N15:238 NXB LEQ N15:238 0 MOV 0 N15:238 NXB GEQ N15:238 16383 MOV 16383 N15:238 BND EOR
%   I:9.7  TEP_BT16  "Teplomer zona 16" %
%   N15:238  "PID skutocna teplota v zone c.16" %
% Rung: 139 %
SOR BST SCP N12:65 -210 760 0 16383 N15:212 NXB LEQ N15:212 0 MOV 0 N15:212 NXB GEQ N15:212 16383 MOV 16383 N15:212 BND EOR
%   N12:65  "Žiadaná teplota v zóne è.16" %
%   N15:212  "PID ziadana teplota v zone c.16" %

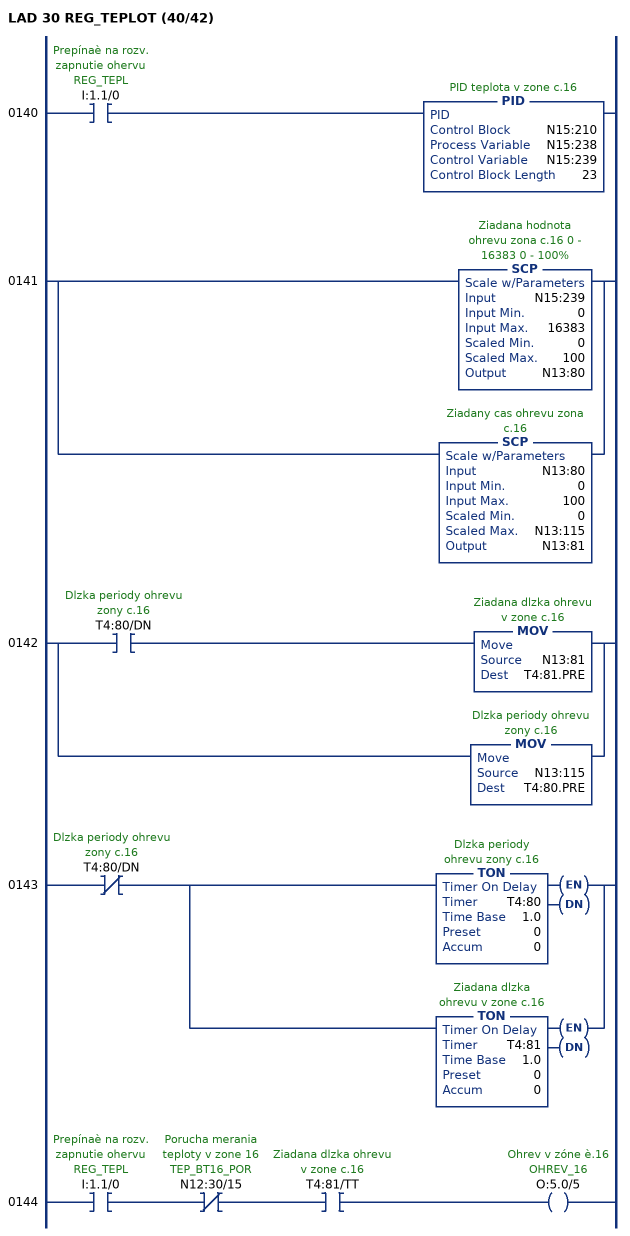
% Rung: 140 %
SOR XIC I:1.1/0 PID N15:210 N15:238 N15:239 23 EOR
%   I:1.1/0  REG_TEPL  "Prepínaè na rozv. zapnutie ohervu" %
%   N15:210  "PID teplota v zone c.16" %
%   N15:238  "PID skutocna teplota v zone c.16" %
% Rung: 141 %
SOR BST SCP N15:239 0 16383 0 100 N13:80 NXB SCP N13:80 0 100 0 N13:115 N13:81 BND EOR
%   N13:80  "Ziadana hodnota ohrevu zona c.16 0 - 16383 0 - 100%" %
%   N13:81  "Ziadany cas ohrevu zona c.16" %
% Rung: 142 %
SOR BST XIC T4:80/DN MOV N13:81 T4:81.PRE NXB MOV N13:115 T4:80.PRE BND EOR
%   T4:80  "Dlzka periody ohrevu zony c.16" %
%   N13:81  "Ziadany cas ohrevu zona c.16" %
%   T4:81  "Ziadana dlzka ohrevu v zone c.16" %
% Rung: 143 %
SOR XIO T4:80/DN BST TON T4:80 1.0 0 0 NXB TON T4:81 1.0 0 0 BND EOR
%   T4:80  "Dlzka periody ohrevu zony c.16" %
%   T4:81  "Ziadana dlzka ohrevu v zone c.16" %
% Rung: 144 %
SOR XIC I:1.1/0 XIO N12:30/15 XIC T4:81/TT OTE O:5.0/5 EOR
%   I:1.1/0  REG_TEPL  "Prepínaè na rozv. zapnutie ohervu" %
%   N12:30/15  TEP_BT16_POR  "Porucha merania teploty v zone 16" %
%   T4:81  "Ziadana dlzka ohrevu v zone c.16" %
%   O:5.0/5  OHREV_16  "Ohrev v zóne è.16" %

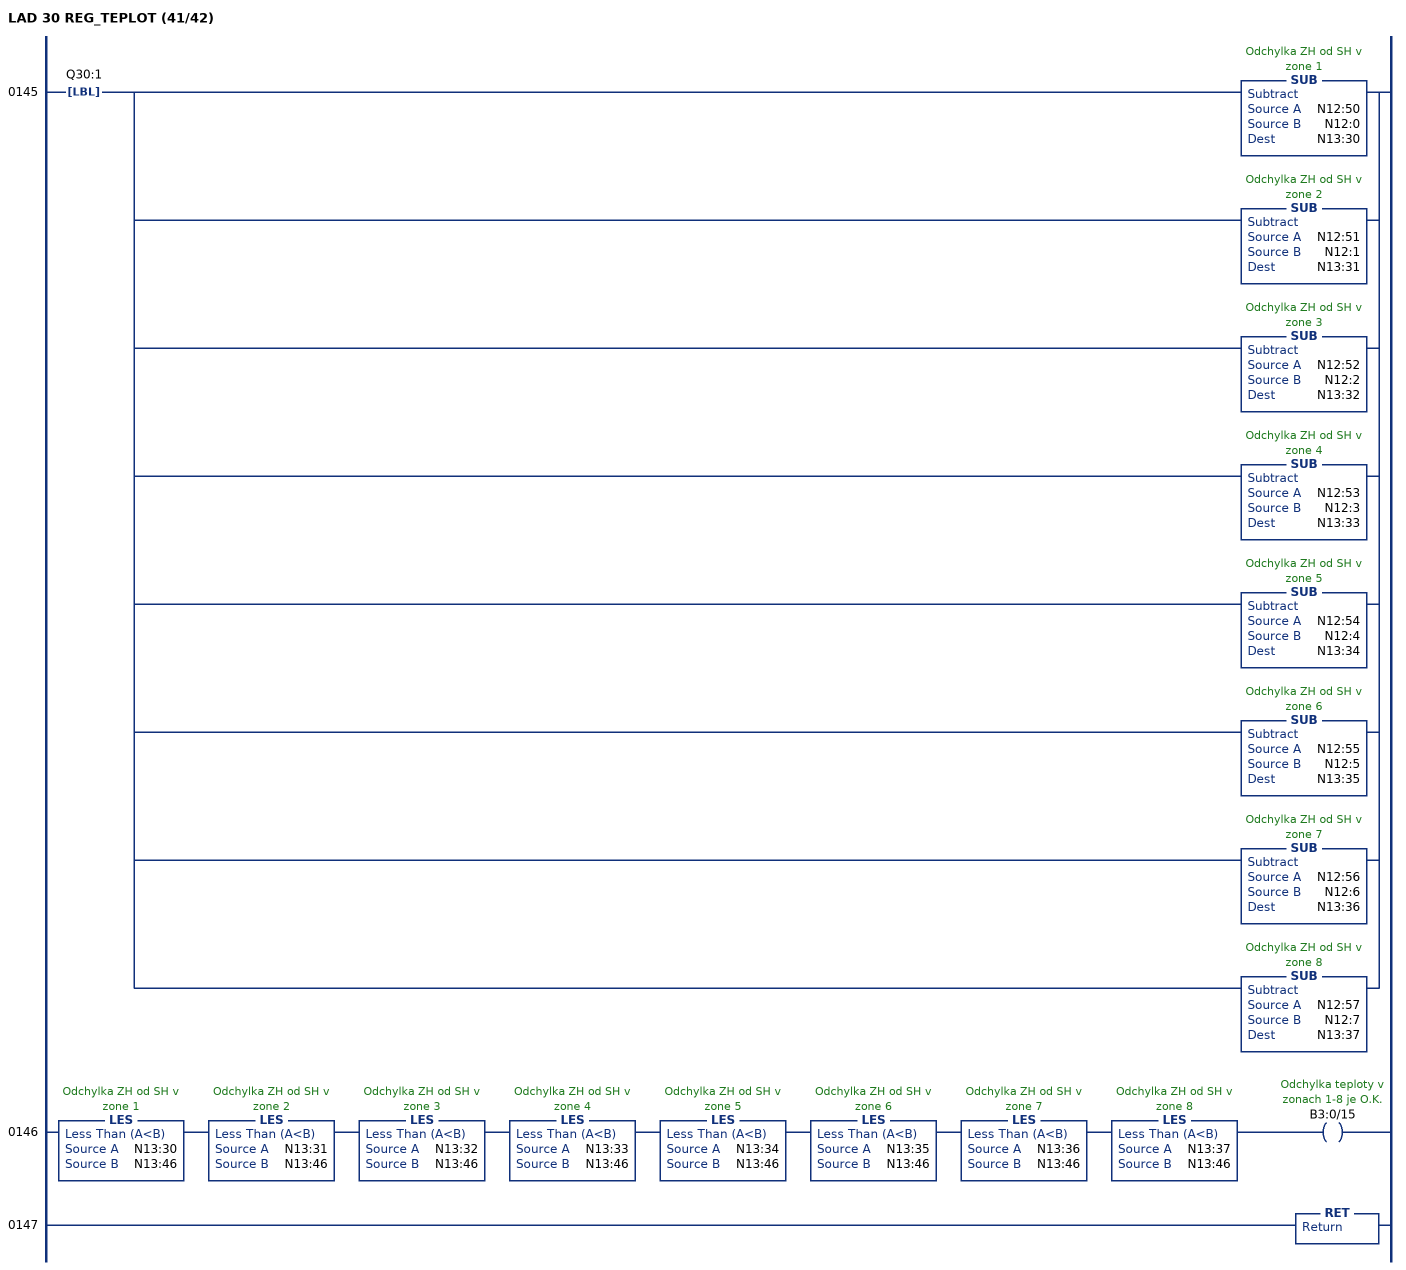
% Rung: 145 %
SOR LBL Q30:1 BST SUB N12:50 N12:0 N13:30 NXB SUB N12:51 N12:1 N13:31 NXB SUB N12:52 N12:2 N13:32 NXB SUB N12:53 N12:3 N13:33 NXB SUB N12:54 N12:4 N13:34 NXB SUB N12:55 N12:5 N13:35 NXB SUB N12:56 N12:6 N13:36 NXB SUB N12:57 N12:7 N13:37 BND EOR
%   N12:50  "Žiadaná teplota v zóne è.1" %
%   N12:0  TEP_Z01  "Teplota v zone 1 185" %
%   N13:30  "Odchylka ZH od SH v zone 1" %
%   N12:51  "Žiadaná teplota v zóne è.2" %
%   N12:1  TEP_Z02  "Teplota v zone 2 190" %
%   N13:31  "Odchylka ZH od SH v zone 2" %
%   N12:52  "Žiadaná teplota v zóne è.3" %
%   N12:2  TEP_Z03  "Teplota v zone 3 190" %
%   N13:32  "Odchylka ZH od SH v zone 3" %
%   N12:53  "Žiadaná teplota v zóne è.4" %
%   N12:3  TEP_Z04  "Teplota v zone 4 195" %
%   N13:33  "Odchylka ZH od SH v zone 4" %
%   N12:54  "Žiadaná teplota v zóne è.5" %
%   N12:4  TEP_Z05  "Teplota v zone 5 195" %
%   N13:34  "Odchylka ZH od SH v zone 5" %
%   N12:55  "Žiadaná teplota v zóne è.6" %
%   N12:5  TEP_Z06  "Teplota v zone 6 195" %
%   N13:35  "Odchylka ZH od SH v zone 6" %
%   N12:56  "Žiadaná teplota v zóne è.7" %
%   N12:6  TEP_Z07  "Teplota v zone 7 195" %
%   N13:36  "Odchylka ZH od SH v zone 7" %
%   N12:57  "Žiadaná teplota v zóne è.8" %
%   N12:7  TEP_Z08  "Teplota v zone 8" %
%   N13:37  "Odchylka ZH od SH v zone 8" %
% Rung: 146 %
SOR LES N13:30 N13:46 LES N13:31 N13:46 LES N13:32 N13:46 LES N13:33 N13:46 LES N13:34 N13:46 LES N13:35 N13:46 LES N13:36 N13:46 LES N13:37 N13:46 OTE B3:0/15 EOR
%   N13:30  "Odchylka ZH od SH v zone 1" %
%   N13:46  "Max velkost odchylky teploty v zonach 1-8" %
%   N13:31  "Odchylka ZH od SH v zone 2" %
%   N13:32  "Odchylka ZH od SH v zone 3" %
%   N13:33  "Odchylka ZH od SH v zone 4" %
%   N13:34  "Odchylka ZH od SH v zone 5" %
%   N13:35  "Odchylka ZH od SH v zone 6" %
%   N13:36  "Odchylka ZH od SH v zone 7" %
%   N13:37  "Odchylka ZH od SH v zone 8" %
%   B3:0/15  "Odchylka teploty v zonach 1-8 je O.K." %
% Rung: 147 %
SOR RET EOR

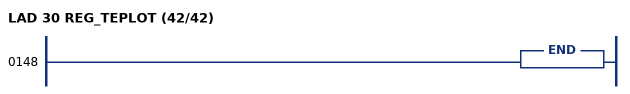
% Rung: 148 %
SOR END EOR

OTHER DOCUMENTED ADDRESSES
  C5:2/DN  NABEH
  C5:3/DN  DOBIHANI
  F9:100  "Žiadané množstvo vody L.Hradok"
  I:1.0/2  CHL_O  "Chlazeni oleje"
  I:1.0/6  AKUMUL  "Akumulator neni vypousten"
  I:1.1/1  "Rezerva"
  I:1.1/2  "Rezerva"
  I:2.0/4  VMD  "Vozik v mezipo- loze dolu"
  I:2.0/6  VMN  "Vozik v mezi- poloze nahoru"
  I:6.1  OT_VS  "Otacky pohonu vytlacov. stroje"
  I:6.5  NI8_REZ1
  I:6.6  NI8_REZ2
  I:6.7  NI8_REZ3
  N7:19  T_10  "Omezeni oddelovani parizonu"
  N7:23  T_14  "Prodleva v uvodu rezimu VYCH.POL."
  N7:25  T_16  "Trvani pulzu blikani"
  N7:26  T_17  "Trvani mezery blikani"
  N7:32  T_23  "Rezerva"
  N7:33  T_24  "Vypnuti hydr.agr. v rezimu VYPNUTO"
  N7:35  T_26  "Zpozdeni hlaseni poruch HA"
  N7:36  T_27  "Prodlou- zeni startu cyklu"
  N7:37  T_28  "Hlidani forem a voziku nahore"
  N7:42  OTACKY  "Otacky sneku vytlacov. stroje"
  N7:43  PROUD  "Proud pohonu vytlacov. stroje"
  N7:44/1  ER_POHON  "Pohon VS neni v chodu"
  N7:44/8  ER_REZERVA  "Puvodne: Neuzavren ventil rizeni"
  N7:47/6  ERROR_VP  "Stroj nebyl ve vychozi poloze"
  N7:50/6  POMOC7
  N7:51/8  REZIM_0
  N7:52/0  ER_M
  N7:52/1  ER_K
  N7:52/2  ER_SM
  N7:52/3  ER_ST
  N7:52/4  ER_H
  N7:52/5  ER_V
  N7:52/6  ER_F
  N7:52/12  ER_VP
  N7:52/14  ER_VN
  N7:53/1  Z45_5
  N7:55/15  L
  N7:56/12  ZM_W13
  N7:56/13  ZM_W14
  N7:60/0  RTS_W1
  N7:60/1  RTS_W2
  N7:60/2  RTS_W3
  N7:60/3  RTS_W4
  N7:60/4  RTS_W5
  N7:60/5  RTS_W6
  N7:62/13  REZ_VP
  N7:68/12  TNP_A
  N7:75/4  POMOC15
  N11:10  DR_K1  "Draha krok 1"
  N11:12  SM_K1  "Smer kroku 1"
  N11:13  START_K1  "Start kroku 1"
  N11:16  SM_K2  "Smer kroku 2"
  N11:17  START_K2  "Start kroku 2"
  N11:22  SM_K3  "Smer kroku 3"
  N11:23  START_K3  "Start kroku 3"
  N11:26  SM_K4  "Smer kroku 4"
  N11:27  START_K4  "Start kroku 4"
  N11:32  SM_K5  "Smer kroku 5"
  N11:33  START_K5  "Start kroku 5"
  N11:34  DR_K6  "Draha kroku 6"
  N11:36  SM_K6  "Smer kroku 6"
  N11:37  START_K6  "Start kroku 6"
  N11:42  SM_K7  "Smer kroku 7"
  N11:43  START_K7  "Start kroku 7"
  N11:46  SM_K8  "Smer kroku 8"
  N11:47  START_K8  "Start kroku 8"
  N11:48  POM_K7
  N11:49  POM_K8
  N11:51  PREP_POL_K1  "Prepocet poloky kroku 1"
  N11:72  SM_VP  "Smer vychozi polohy"
  N11:75  POL_VP
  N11:80  POV_K2
  N11:81  POV_K3
  N11:82  POV_K4
  N11:83  POV_K5
  N11:84  POV_K6
  N11:90/1  K1_STAT
  N11:90/6  K6_STAT
  N11:90/7  K7_STAT
  N11:90/8  K8_STAT
  N12:78  "Dolná hranica teploty v zóne è.9"
  N12:79  "Dolná hranica teploty v zóne è.10"
  N12:80  "Dolná hranica teploty v zóne è.11"
  N12:81  "Dolná hranica teploty v zóne è.12"
  N12:82  "Dolná hranica teploty v zóne è.13"
  N12:83  "Dolná hranica teploty v zóne è.14"
  N12:84  "Dolná hranica teploty v zóne è.15"
  N12:85  "Dolná hranica teploty v zóne è.16"
  N12:98  "Horná hranica teploty v zóne è.9"
  N12:99  "Horná hranica teploty v zóne è.10"
  N12:100  "Horná hranica teploty v zóne è.11"
  N12:101  "Horná hranica teploty v zóne è.12"
  N12:102  "Horná hranica teploty v zóne è.13"
  N12:103  "Horná hranica teploty v zóne è.14"
  N12:104  "Horná hranica teploty v zóne è.15"
  N12:105  "Horná hranica teploty v zóne è.16"
  N12:154  "Žiadaná rýchlost vozíka c.2 dolu"
  N12:155  "Žiadaná rýchlost vozíka c.3 dolu"
  N13:50  "Ziadana hodnota ohrevu zona c.1 0 - 16383 0 - 100%"
  N13:52  "Ziadana hodnota ohrevu zona c.2 0 - 16383 0 - 100%"
  N13:54  "Ziadana hodnota ohrevu zona c.3 0 - 16383 0 - 100%"
  N13:56  "Ziadana hodnota ohrevu zona c.4 0 - 16383 0 - 100%"
  N13:58  "Ziadana hodnota ohrevu zona c.5 0 - 16383 0 - 100%"
  N13:60  "Ziadana hodnota ohrevu zona c.6 0 - 16383 0 - 100%"
  N13:62  "Ziadana hodnota ohrevu zona c.7 0 - 16383 0 - 100%"
  N13:64  "Ziadana hodnota ohrevu zona c.8 0 - 16383 0 - 100%"
  O:4.0/0  VNR  "Vozik nahoru rychle"
  O:4.0/1  VNP  "Vozik nahoru pomalu"
  O:4.0/2  VDR  "Vozik dolu rychle"
  O:4.0/3  VDP  "Vozik dolu pomalu"
  O:5.0/9  CHLAD_2  "Chladenie v zóne è.2"
  O:5.0/10  OHREV_3  "Ohrev v zóne è.3"
  O:7.0/10  TDR
  O:7.0/11  TDP
  O:7.0/12  TNR
  O:7.0/13  TNP

COMMENTS NOT ATTACHED TO A CURRENT RUNG
  N10:251: Podprogram pro praci s archivnimi kopiemi receptur 1 - 8.
    Archivni kopie receptur jsou ve file N10:00 - N10:239 (8 x 30 slov).
    Prenosy receptur z archivnich kopii 1 - 8 d/z aktualni receptury musi povolit
    hlavni program nastavenim REC_ENABLE=1.
    
                           Prace s archivnimi kopiemi receptur zakazana:
  N10:253: Prace s archivnimi kopiemi receptur povolena:
  N7:50/7: DIAGNOSTIKA NAJETI STROJE DO VYCHOZI POLOHY:

REVISION NOTES
  0: Roysireni programu o analogove rizeni ventilu vyfukovaciho trnu

DATA TABLE (non-zero values as saved)
DATA B3
% B3:0 % 0X8402 0X0012
DATA T4
% .PRE .ACC %
% T4:0 % 6000 0
% T4:1 % 6000 0
% T4:2 % 4500 0
% T4:3 % 210 0
% T4:4 % 5500 0
% T4:5 % 95 0
% T4:7 % 5000 0
% T4:8 % 990 0
% T4:9 % 90 0
% T4:10 % 400 0
% T4:11 % 60 0
% T4:13 % 350 0
% T4:14 % 400 400
% T4:16 % 40 41
% T4:17 % 40 39
% T4:22 % 90 0
% T4:23 % 2000 0
% T4:24 % 500 0
% T4:25 % 50 0
% T4:26 % 2000 0
% T4:27 % 50 50
% T4:28 % 15000 0
% T4:35 % 40 0
% T4:36 % 40 0
% T4:37 % 50 0
% T4:50 % 1000 65
% T4:51 % 432 65
% T4:52 % 500 331
% T4:53 % 354 342
% T4:54 % 1000 76
% T4:55 % 209 76
% T4:56 % 500 461
% T4:57 % 104 104
% T4:58 % 500 328
% T4:59 % 149 149
% T4:60 % 500 328
% T4:61 % 253 253
% T4:62 % 500 344
% T4:63 % 334 335
% T4:64 % 500 237
% T4:65 % 499 237
% T4:66 % 10 0
% T4:67 % 1 0
% T4:68 % 10 0
% T4:69 % 1 0
% T4:70 % 10 0
% T4:71 % 1 0
DATA C5
% .PRE .ACC %
% C5:0 % 30000 904
% C5:1 % 10000 -14841
% C5:2 % 30000 0
% C5:3 % 10 0
% C5:4 % 1000 999
DATA N7
% N7:0 % 1500 0 0 0 0 0 0 0 4352 6000
% N7:10 % 6000 4500 210 5500 95 0 5000 990 90 200
% N7:20 % 60 0 350 300 0 40 40 0 0 0
% N7:30 % 0 90 1700 500 50 500 50 400 0 0
% N7:40 % 0 10000 0 0 -32768 0 0 0 8 0
% N7:50 % 8195 64 0 -28248 32 0 512 16385 8192 68
% N7:60 % 0 0 7935 0 0 0 0 0 0 0
% N7:70 % -3152 -4927 0 0 0 -32636 71 0 0 0
% N7:80 % 750 5 100 0 100 10 0 0 0 0
% N7:90 % 1893 0 0 0 0 0 0 0
DATA F8
% F8:0 % 0 0 5.679e+07 5.679e+07 5.679e+07
% F8:5 % 5.679e+07 0 0 0 0
DATA N9
% N9:0 % 5 5 5 5 5 5 5 5 0 0
DATA N10
% N10:0 % 5000 500 4300 200 4000 200 20 4500 400 20
% N10:10 % 200 20 20 150 300 50 200 400 600 800
% N10:30 % 5000 500 4300 200 4000 200 20 4500 400 20
% N10:40 % 200 20 20 150 300 50 200 400 600 800
% N10:60 % 1500 1500 1350 200 900 350 20 1300 100 20
% N10:70 % 200 20 20 110 300 50 200 400 600 800
% N10:90 % 1500 500 100 300 900 200 20 1300 150 20
% N10:100 % 200 20 20 150 300 50 200 400 600 800
% N10:120 % 1500 500 100 300 900 200 20 1300 150 20
% N10:130 % 200 20 20 150 300 50 200 400 600 800
% N10:150 % 1500 500 100 300 900 200 20 1300 150 20
% N10:160 % 200 20 20 150 300 50 200 400 600 800
% N10:180 % 1500 500 100 300 900 200 20 1300 150 20
% N10:190 % 200 20 20 150 300 50 200 400 600 800
% N10:210 % 1500 500 100 300 900 200 20 1300 150 20
% N10:220 % 200 20 20 150 300 50 200 400 600 800
% N10:250 % 2 2 1 2 1 0
DATA N11
% N11:10 % 0 60 0 0 940 75 0 0 0 0
% N11:20 % 930 25 1 0 900 0 0 0 0 0
% N11:30 % 190 90 0 0 107 90 1 0 0 0
% N11:40 % 100 30 1 0 948 40 0 0 0 0
% N11:50 % -19661 0 -24576 947 8192 928 0 955 0 0
% N11:60 % 29490 926 29490 150 9830 135 -13107 601 135 0
% N11:70 % 789 9830 1 0 30 0 1003 1002 0 0
% N11:90 % 0 1 0 0 0 0 0 0 0 0
% N11:100 % 7077 11587 3417 3441 4881 8301 10959 16368 0 0
DATA N12
% N12:0 % 190 192 185 191 195 200 199 40 -210 -210
% N12:10 % -210 -210 -210 -210 -210 -210 0 0 0 0
% N12:50 % 190 195 190 195 195 200 200 40 0 0
% N12:70 % 192 197 192 197 195 200 200 42 -1 -1
% N12:80 % -1 -1 -1 -1 -1 -1 0 0 0 0
% N12:90 % 194 199 194 199 196 201 201 44 1 1
% N12:100 % 1 1 1 1 1 1 0 0 0 0
% N12:120 % 1010 800 400 60 30 0 0 0 0 0
% N12:130 % 0 150 600 950 980 100 0 0 0 0
% N12:150 % 30 80 45 30 0 0 0 30 0 0
% N12:160 % 80 45 35 30 0 0 30 0 0 0
% N12:170 % 41 0 0 0 0 20 0 0 0 0
% N12:180 % 0 100 600 700 900 100 0 0 0 0
% N12:190 % 70 50 35 30 0 0 0 0 0 0
% N12:200 % 1010 810 800 600 10 0 0 0 0 0
% N12:210 % 40 20 40 30 0 25 30 0 0 0
DATA N13
% N13:0 % -32703 -32703 -32703 -32703 -32703 -32703 -32703 -32703 0 -32703
% N13:10 % -32703 -32703 -32703 -32703 -32703 -32703 -32703 2048 2048 2048
% N13:20 % 2048 2048 2048 2048 2048 0 0 0 0 0
% N13:30 % 0 3 5 4 0 0 1 0 0 0
% N13:40 % 0 0 0 0 0 0 20 0 0 0
% N13:50 % 7 432 178 353 3 209 4 105 3 149
% N13:60 % 3 253 14 334 3 500 10 1 12 1
% N13:70 % 12 1 12 0 12 0 12 0 12 0
% N13:80 % 12 0 0 0 0 0 0 0 0 0
% N13:100 % 1000 500 1000 500 500 500 500 500 10 10
% N13:110 % 10 0 0 0 0 0 0 0 0 0
% N13:120 % 0 20 80 90 95 100 0 0 0 0
% N13:200 % 0 20 55 70 85 100 0 0 0 0
DATA N14
% N14:0 % -24503 0 6756 5 10 0 0 16383 0 0
% N14:10 % 0 100 0 1 6748 8 43 7072 27409 1
% N14:20 % -23104 14054 6756 0 0 0 0 0 6748 7076
% N14:30 % -24503 0 6840 100 50 0 0 16383 0 0
% N14:40 % 0 100 10 1 6789 51 71 11069 -15640 1
% N14:50 % -22448 14055 6840 0 0 0 0 0 6789 11579
% N14:60 % -24503 0 6756 7 10 0 0 16383 0 0
% N14:70 % 0 100 10 1 6676 80 21 3363 2751 1
% N14:80 % -24256 11575 6756 0 0 0 0 0 6676 3419
% N14:90 % -32759 0 6840 100 50 0 0 16383 0 0
% N14:100 % 0 100 10 10 6774 66 21 2796 2148 1
% N14:110 % -22688 8264 6840 0 0 0 0 0 6774 3456
% N14:120 % -32759 0 6840 120 50 0 0 16383 0 0
% N14:130 % 0 100 10 10 6836 4 30 4845 29040 1
% N14:140 % -21696 8425 6840 0 0 0 0 0 6836 4893
% N14:150 % -32759 0 6925 100 50 0 0 16383 0 0
% N14:160 % 0 100 10 10 6917 8 51 8232 -30020 1
% N14:170 % -20400 8586 6925 0 0 0 0 0 6917 8312
% N14:180 % -24503 0 6925 100 100 0 0 16383 0 0
% N14:190 % 0 100 10 1 6908 17 67 10790 30003 1
% N14:200 % -20544 14122 6925 0 0 0 0 0 6908 10960
% N14:210 % -24503 0 4222 100 100 0 0 16383 0 0
% N14:220 % 0 100 10 1 4215 7 100 16298 -30981 1
% N14:230 % 1904 14123 4222 0 0 0 0 0 4215 16368
DATA N15
% N15:0 % 1 0 3547 1 10 0 0 16383 0 0
% N15:10 % 0 100 0 1023 0 0 0 0 0 0
% N15:20 % 0 0 0 0 0 0 0 0 0 1632
% N15:30 % 1 0 3547 1 10 0 0 16383 0 0
% N15:40 % 0 100 0 1000 0 0 0 0 0 0
% N15:50 % 0 0 0 0 0 0 0 0 0 1961
% N15:60 % 1 0 3547 1 10 0 0 16383 0 0
% N15:70 % 0 100 0 1000 0 0 0 0 0 0
% N15:80 % 0 0 0 0 0 0 0 0 0 1961
% N15:90 % 1 0 3547 1 10 0 0 16383 0 0
% N15:100 % 0 100 0 1000 0 0 0 0 0 0
% N15:110 % 0 0 0 0 0 0 0 0 0 1961
% N15:120 % 1 0 3547 1 10 0 0 16383 0 0
% N15:130 % 0 100 0 1000 0 0 0 0 0 0
% N15:140 % 0 0 0 0 0 0 0 0 0 1961
% N15:150 % 1 0 3547 1 10 0 0 16383 0 0
% N15:160 % 0 100 0 1000 0 0 0 0 0 0
% N15:170 % 0 0 0 0 0 0 0 0 0 1961
% N15:180 % 1 0 3547 1 10 0 0 16383 0 0
% N15:190 % 0 100 0 1000 0 0 0 0 0 0
% N15:200 % 0 0 0 0 0 0 0 0 0 1961
% N15:210 % 1 0 3547 1 10 0 0 16383 0 0
% N15:220 % 0 100 0 1000 0 0 0 0 0 0
% N15:230 % 0 0 0 0 0 0 0 0 0 1961
